	STP.P210A3_LimePumpS1_LocalRemoteStat AT %IX259.1 : BOOL;	(*  ~ {LinkedWith:TIID^C6920 (EtherCAT)^ScadaRoom_KouplerUTP (EK1100)^ScadaRoom_KouplerFiber (EK1521)^ChemicalAndTertiary (EK1501)^Term 90 (EL1809) A9^Channel 3^Input} *)
	STP.P203A_LimeCirculationPump1_LocalRemoteStat AT %IX111.1 : BOOL;	(*  ~ {LinkedWith:TIID^C6920 (EtherCAT)^ScadaRoom_KouplerUTP (EK1100)^ScadaRoom_KouplerFiber (EK1521)^ChemicalAndTertiary (EK1501)^Term 90 (EL1809) A9^Channel 6^Input} *)
	STP.P203B_LimeCirculationPump2_LocalRemoteStat AT %IX259.2 : BOOL;	(*  ~ {LinkedWith:TIID^C6920 (EtherCAT)^ScadaRoom_KouplerUTP (EK1100)^ScadaRoom_KouplerFiber (EK1521)^ChemicalAndTertiary (EK1501)^Term 90 (EL1809) A9^Channel 7^Input} *)
	STP.P211A1_AlumPumpSBRS1_LocalRemoteStat AT %IX96.1 : BOOL;	(*  ~ {LinkedWith:TIID^C6920 (EtherCAT)^ScadaRoom_KouplerUTP (EK1100)^ScadaRoom_KouplerFiber (EK1521)^ChemicalAndTertiary (EK1501)^Term 90 (EL1809) A9^Channel 8^Input} *)
	STP.P211A2_AlumPumpSBRS1_LocalRemoteStat AT %IX96.2 : BOOL;	(*  ~ {LinkedWith:TIID^C6920 (EtherCAT)^ScadaRoom_KouplerUTP (EK1100)^ScadaRoom_KouplerFiber (EK1521)^ChemicalAndTertiary (EK1501)^Term 90 (EL1809) A9^Channel 9^Input} *)
	STP.P211B1_AlumPumpSBRS2_LocalRemoteStat AT %IX96.3 : BOOL;	(*  ~ {LinkedWith:TIID^C6920 (EtherCAT)^ScadaRoom_KouplerUTP (EK1100)^ScadaRoom_KouplerFiber (EK1521)^ChemicalAndTertiary (EK1501)^Term 90 (EL1809) A9^Channel 10^Input} *)
	STP.P211B2_AlumPump2SBRS2_LocalRemoteStat AT %IX96.4 : BOOL;	(*  ~ {LinkedWith:TIID^C6920 (EtherCAT)^ScadaRoom_KouplerUTP (EK1100)^ScadaRoom_KouplerFiber (EK1521)^ChemicalAndTertiary (EK1501)^Term 90 (EL1809) A9^Channel 11^Input} *)
	STP.P352A_AlumPumpTertiaryDosing_LocalRemoteStat AT %IX111.2 : BOOL;	(*  ~ {LinkedWith:TIID^C6920 (EtherCAT)^ScadaRoom_KouplerUTP (EK1100)^ScadaRoom_KouplerFiber (EK1521)^ChemicalAndTertiary (EK1501)^Term 90 (EL1809) A9^Channel 12^Input} *)
	STP.P352B_AlumPumpTertiaryDosing_LocalRemoteStat AT %IX111.3 : BOOL;	(*  ~ {LinkedWith:TIID^C6920 (EtherCAT)^ScadaRoom_KouplerUTP (EK1100)^ScadaRoom_KouplerFiber (EK1521)^ChemicalAndTertiary (EK1501)^Term 90 (EL1809) A9^Channel 13^Input} *)
	STP.P354A_CausticSodaPump_LocalRemoteStat AT %IX111.4 : BOOL;	(*  ~ {LinkedWith:TIID^C6920 (EtherCAT)^ScadaRoom_KouplerUTP (EK1100)^ScadaRoom_KouplerFiber (EK1521)^ChemicalAndTertiary (EK1501)^Term 90 (EL1809) A9^Channel 14^Input} *)
	STP.P354B_CausticSodaPump_LocalRemoteStat AT %IX111.5 : BOOL;	(*  ~ {LinkedWith:TIID^C6920 (EtherCAT)^ScadaRoom_KouplerUTP (EK1100)^ScadaRoom_KouplerFiber (EK1521)^ChemicalAndTertiary (EK1501)^Term 90 (EL1809) A9^Channel 15^Input} *)
	STP.P356A_SodiumHypochloritePump_LocalRemoteStat AT %IX112.0 : BOOL;	(*  ~ {LinkedWith:TIID^C6920 (EtherCAT)^ScadaRoom_KouplerUTP (EK1100)^ScadaRoom_KouplerFiber (EK1521)^ChemicalAndTertiary (EK1501)^Term 91 (EL1809) A10^Channel 3^Input} *)
	STP.P356B_SodiumHypochloritePump_LocalRemoteStat AT %IX112.1 : BOOL;	(*  ~ {LinkedWith:TIID^C6920 (EtherCAT)^ScadaRoom_KouplerUTP (EK1100)^ScadaRoom_KouplerFiber (EK1521)^ChemicalAndTertiary (EK1501)^Term 91 (EL1809) A10^Channel 4^Input} *)
	STP.P301A_EffluentTransferPump_LocalRemoteStat AT %IX112.2 : BOOL;	(*  ~ {LinkedWith:TIID^C6920 (EtherCAT)^ScadaRoom_KouplerUTP (EK1100)^ScadaRoom_KouplerFiber (EK1521)^ChemicalAndTertiary (EK1501)^Term 91 (EL1809) A10^Channel 5^Input} *)
	STP.P301B_EffluentTransferPump_LocalRemoteStat AT %IX112.3 : BOOL;	(*  ~ {LinkedWith:TIID^C6920 (EtherCAT)^ScadaRoom_KouplerUTP (EK1100)^ScadaRoom_KouplerFiber (EK1521)^ChemicalAndTertiary (EK1501)^Term 91 (EL1809) A10^Channel 6^Input} *)
	STP.P302A_CollectionPump_LocalRemoteStat AT %IX112.4 : BOOL;	(*  ~ {LinkedWith:TIID^C6920 (EtherCAT)^ScadaRoom_KouplerUTP (EK1100)^ScadaRoom_KouplerFiber (EK1521)^ChemicalAndTertiary (EK1501)^Term 91 (EL1809) A10^Channel 7^Input} *)
	STP.P302B_CollectionPump_LocalRemoteStat AT %IX112.5 : BOOL;	(*  ~ {LinkedWith:TIID^C6920 (EtherCAT)^ScadaRoom_KouplerUTP (EK1100)^ScadaRoom_KouplerFiber (EK1521)^ChemicalAndTertiary (EK1501)^Term 91 (EL1809) A10^Channel 8^Input} *)
	STP.K301A_AirCompressor_LocalRemoteStat AT %IX112.6 : BOOL;	(*  ~ {LinkedWith:TIID^C6920 (EtherCAT)^ScadaRoom_KouplerUTP (EK1100)^ScadaRoom_KouplerFiber (EK1521)^ChemicalAndTertiary (EK1501)^Term 91 (EL1809) A10^Channel 9^Input} *)
	STP.K301B_AirCompressor_LocalRemoteStat AT %IX112.7 : BOOL;	(*  ~ {LinkedWith:TIID^C6920 (EtherCAT)^ScadaRoom_KouplerUTP (EK1100)^ScadaRoom_KouplerFiber (EK1521)^ChemicalAndTertiary (EK1501)^Term 91 (EL1809) A10^Channel 10^Input} *)
	STP.M210A_LimeStirrer_LocalRemoteStat AT %IX288.0 : BOOL;	(*  ~ {LinkedWith:TIID^C6920 (EtherCAT)^ScadaRoom_KouplerUTP (EK1100)^ScadaRoom_KouplerFiber (EK1521)^ChemicalAndTertiary (EK1501)^Term 91 (EL1809) A10^Channel 11^Input} *)
	STP.M210B_LimeStirrer_LocalRemoteStat AT %IX288.1 : BOOL;	(*  ~ {LinkedWith:TIID^C6920 (EtherCAT)^ScadaRoom_KouplerUTP (EK1100)^ScadaRoom_KouplerFiber (EK1521)^ChemicalAndTertiary (EK1501)^Term 91 (EL1809) A10^Channel 12^Input} *)
	STP.M210C_LimeStirrer_LocalRemoteStat AT %IX288.2 : BOOL;	(*  ~ {LinkedWith:TIID^C6920 (EtherCAT)^ScadaRoom_KouplerUTP (EK1100)^ScadaRoom_KouplerFiber (EK1521)^ChemicalAndTertiary (EK1501)^Term 91 (EL1809) A10^Channel 13^Input} *)
	STP.P210A1_LimePumpS1_TripStat AT %IX113.0 : BOOL;	(*  ~ {LinkedWith:TIID^C6920 (EtherCAT)^ScadaRoom_KouplerUTP (EK1100)^ScadaRoom_KouplerFiber (EK1521)^ChemicalAndTertiary (EK1501)^Term 92 (EL1809) A11^Channel 1^Input} *)
	STP.P210A2_LimePumpS1_TripStat AT %IX113.1 : BOOL;	(*  ~ {LinkedWith:TIID^C6920 (EtherCAT)^ScadaRoom_KouplerUTP (EK1100)^ScadaRoom_KouplerFiber (EK1521)^ChemicalAndTertiary (EK1501)^Term 92 (EL1809) A11^Channel 2^Input} *)
	STP.P210A3_LimePumpS1_TripStat AT %IX113.2 : BOOL;	(*  ~ {LinkedWith:TIID^C6920 (EtherCAT)^ScadaRoom_KouplerUTP (EK1100)^ScadaRoom_KouplerFiber (EK1521)^ChemicalAndTertiary (EK1501)^Term 92 (EL1809) A11^Channel 3^Input} *)
	STP.P203A_LimeCirculationPump_TripStat AT %IX113.3 : BOOL;	(*  ~ {LinkedWith:TIID^C6920 (EtherCAT)^ScadaRoom_KouplerUTP (EK1100)^ScadaRoom_KouplerFiber (EK1521)^ChemicalAndTertiary (EK1501)^Term 92 (EL1809) A11^Channel 6^Input} *)
	STP.P203B_LimeCirculationPump_TripStat AT %IX113.4 : BOOL;	(*  ~ {LinkedWith:TIID^C6920 (EtherCAT)^ScadaRoom_KouplerUTP (EK1100)^ScadaRoom_KouplerFiber (EK1521)^ChemicalAndTertiary (EK1501)^Term 92 (EL1809) A11^Channel 7^Input} *)
	STP.P211A1_AlumPumpSBRS1_TripStat AT %IX113.5 : BOOL;	(*  ~ {LinkedWith:TIID^C6920 (EtherCAT)^ScadaRoom_KouplerUTP (EK1100)^ScadaRoom_KouplerFiber (EK1521)^ChemicalAndTertiary (EK1501)^Term 92 (EL1809) A11^Channel 8^Input} *)
	STP.P211A2_AlumPumpSBRS1_TripStat AT %IX113.6 : BOOL;	(*  ~ {LinkedWith:TIID^C6920 (EtherCAT)^ScadaRoom_KouplerUTP (EK1100)^ScadaRoom_KouplerFiber (EK1521)^ChemicalAndTertiary (EK1501)^Term 92 (EL1809) A11^Channel 9^Input} *)
	STP.P211B1_AlumPumpSBRS1_TripStat AT %IX113.7 : BOOL;	(*  ~ {LinkedWith:TIID^C6920 (EtherCAT)^ScadaRoom_KouplerUTP (EK1100)^ScadaRoom_KouplerFiber (EK1521)^ChemicalAndTertiary (EK1501)^Term 92 (EL1809) A11^Channel 10^Input} *)
	STP.P211B2_AlumPumpSBRS2_TripStat AT %IX114.0 : BOOL;	(*  ~ {LinkedWith:TIID^C6920 (EtherCAT)^ScadaRoom_KouplerUTP (EK1100)^ScadaRoom_KouplerFiber (EK1521)^ChemicalAndTertiary (EK1501)^Term 92 (EL1809) A11^Channel 11^Input} *)
	STP.P352A_AlumPumpTertiaryDosing_TripStat AT %IX114.1 : BOOL;	(*  ~ {LinkedWith:TIID^C6920 (EtherCAT)^ScadaRoom_KouplerUTP (EK1100)^ScadaRoom_KouplerFiber (EK1521)^ChemicalAndTertiary (EK1501)^Term 92 (EL1809) A11^Channel 12^Input} *)
	STP.P352B_AlumPumpTertiaryDosing_TripStat AT %IX114.2 : BOOL;	(*  ~ {LinkedWith:TIID^C6920 (EtherCAT)^ScadaRoom_KouplerUTP (EK1100)^ScadaRoom_KouplerFiber (EK1521)^ChemicalAndTertiary (EK1501)^Term 92 (EL1809) A11^Channel 13^Input} *)
	STP.P354A_CausticSodaPump_TripStat AT %IX114.3 : BOOL;	(*  ~ {LinkedWith:TIID^C6920 (EtherCAT)^ScadaRoom_KouplerUTP (EK1100)^ScadaRoom_KouplerFiber (EK1521)^ChemicalAndTertiary (EK1501)^Term 92 (EL1809) A11^Channel 14^Input} *)
	STP.P354B_CausticSodaPump_TripStat AT %IX114.4 : BOOL;	(*  ~ {LinkedWith:TIID^C6920 (EtherCAT)^ScadaRoom_KouplerUTP (EK1100)^ScadaRoom_KouplerFiber (EK1521)^ChemicalAndTertiary (EK1501)^Term 92 (EL1809) A11^Channel 15^Input} *)
	STP.P356A_SodiumHypochloritePump_TripStat AT %IX114.7 : BOOL;	(*  ~ {LinkedWith:TIID^C6920 (EtherCAT)^ScadaRoom_KouplerUTP (EK1100)^ScadaRoom_KouplerFiber (EK1521)^ChemicalAndTertiary (EK1501)^Term 93 (EL1809) A12^Channel 3^Input} *)
	STP.P356B_SodiumHypochloritePump_TripStat AT %IX115.0 : BOOL;	(*  ~ {LinkedWith:TIID^C6920 (EtherCAT)^ScadaRoom_KouplerUTP (EK1100)^ScadaRoom_KouplerFiber (EK1521)^ChemicalAndTertiary (EK1501)^Term 93 (EL1809) A12^Channel 4^Input} *)
	STP.P301A_EffluentTransferPump_TripStat AT %IX115.1 : BOOL;	(*  ~ {LinkedWith:TIID^C6920 (EtherCAT)^ScadaRoom_KouplerUTP (EK1100)^ScadaRoom_KouplerFiber (EK1521)^ChemicalAndTertiary (EK1501)^Term 93 (EL1809) A12^Channel 5^Input} *)
	STP.P301B_EffluentTransferPump_TripStat AT %IX115.2 : BOOL;	(*  ~ {LinkedWith:TIID^C6920 (EtherCAT)^ScadaRoom_KouplerUTP (EK1100)^ScadaRoom_KouplerFiber (EK1521)^ChemicalAndTertiary (EK1501)^Term 93 (EL1809) A12^Channel 6^Input} *)
	STP.P302A_CollectionPump_TripStat AT %IX115.3 : BOOL;	(*  ~ {LinkedWith:TIID^C6920 (EtherCAT)^ScadaRoom_KouplerUTP (EK1100)^ScadaRoom_KouplerFiber (EK1521)^ChemicalAndTertiary (EK1501)^Term 93 (EL1809) A12^Channel 7^Input} *)
	STP.P302B_CollectionPump_TripStat AT %IX115.4 : BOOL;	(*  ~ {LinkedWith:TIID^C6920 (EtherCAT)^ScadaRoom_KouplerUTP (EK1100)^ScadaRoom_KouplerFiber (EK1521)^ChemicalAndTertiary (EK1501)^Term 93 (EL1809) A12^Channel 8^Input} *)
	STP.K301A_AirCompressor_TripStat AT %IX115.5 : BOOL;	(*  ~ {LinkedWith:TIID^C6920 (EtherCAT)^ScadaRoom_KouplerUTP (EK1100)^ScadaRoom_KouplerFiber (EK1521)^ChemicalAndTertiary (EK1501)^Term 93 (EL1809) A12^Channel 9^Input} *)
	STP.K301B_AirCompressor_TripStat AT %IX115.6 : BOOL;	(*  ~ {LinkedWith:TIID^C6920 (EtherCAT)^ScadaRoom_KouplerUTP (EK1100)^ScadaRoom_KouplerFiber (EK1521)^ChemicalAndTertiary (EK1501)^Term 93 (EL1809) A12^Channel 10^Input} *)
	STP.M303A_Floculator_TripStat AT %IX259.3 : BOOL;	(*  ~ {LinkedWith:TIID^C6920 (EtherCAT)^ScadaRoom_KouplerUTP (EK1100)^ScadaRoom_KouplerFiber (EK1521)^ChemicalAndTertiary (EK1501)^Term 93 (EL1809) A12^Channel 11^Input} *)
	STP.M303B_Floculator_TripStat AT %IX259.4 : BOOL;	(*  ~ {LinkedWith:TIID^C6920 (EtherCAT)^ScadaRoom_KouplerUTP (EK1100)^ScadaRoom_KouplerFiber (EK1521)^ChemicalAndTertiary (EK1501)^Term 93 (EL1809) A12^Channel 12^Input} *)
	STP.M303C_Floculator_TripStat AT %IX259.5 : BOOL;	(*  ~ {LinkedWith:TIID^C6920 (EtherCAT)^ScadaRoom_KouplerUTP (EK1100)^ScadaRoom_KouplerFiber (EK1521)^ChemicalAndTertiary (EK1501)^Term 93 (EL1809) A12^Channel 13^Input} *)
	STP.M303D_Floculator_TripStat AT %IX259.6 : BOOL;	(*  ~ {LinkedWith:TIID^C6920 (EtherCAT)^ScadaRoom_KouplerUTP (EK1100)^ScadaRoom_KouplerFiber (EK1521)^ChemicalAndTertiary (EK1501)^Term 93 (EL1809) A12^Channel 14^Input} *)
	STP.P210A1_LimePumpS1_EStopStat AT %IX259.7 : BOOL;	(*  ~ {LinkedWith:TIID^C6920 (EtherCAT)^ScadaRoom_KouplerUTP (EK1100)^ScadaRoom_KouplerFiber (EK1521)^ChemicalAndTertiary (EK1501)^Term 94 (EL1809) A13^Channel 1^Input} *)
	STP.P210A2_LimePumpS1_EStopStat AT %IX260.0 : BOOL;	(*  ~ {LinkedWith:TIID^C6920 (EtherCAT)^ScadaRoom_KouplerUTP (EK1100)^ScadaRoom_KouplerFiber (EK1521)^ChemicalAndTertiary (EK1501)^Term 94 (EL1809) A13^Channel 2^Input} *)
	STP.P210A3_LimePumpS1_EStopStat AT %IX260.1 : BOOL;	(*  ~ {LinkedWith:TIID^C6920 (EtherCAT)^ScadaRoom_KouplerUTP (EK1100)^ScadaRoom_KouplerFiber (EK1521)^ChemicalAndTertiary (EK1501)^Term 94 (EL1809) A13^Channel 3^Input} *)
	STP.P203A_LimeCirculationPump_EStopStat AT %IX260.2 : BOOL;	(*  ~ {LinkedWith:TIID^C6920 (EtherCAT)^ScadaRoom_KouplerUTP (EK1100)^ScadaRoom_KouplerFiber (EK1521)^ChemicalAndTertiary (EK1501)^Term 94 (EL1809) A13^Channel 6^Input} *)
	STP.P203B_LimeCirculationPump_EStopStat AT %IX260.3 : BOOL;	(*  ~ {LinkedWith:TIID^C6920 (EtherCAT)^ScadaRoom_KouplerUTP (EK1100)^ScadaRoom_KouplerFiber (EK1521)^ChemicalAndTertiary (EK1501)^Term 94 (EL1809) A13^Channel 7^Input} *)
	STP.P211A1_AlumPumpSBRS1_EStopStat AT %IX260.4 : BOOL;	(*  ~ {LinkedWith:TIID^C6920 (EtherCAT)^ScadaRoom_KouplerUTP (EK1100)^ScadaRoom_KouplerFiber (EK1521)^ChemicalAndTertiary (EK1501)^Term 94 (EL1809) A13^Channel 8^Input} *)
	STP.P211A2_AlumPumpSBRS1_EStopStat AT %IX260.5 : BOOL;	(*  ~ {LinkedWith:TIID^C6920 (EtherCAT)^ScadaRoom_KouplerUTP (EK1100)^ScadaRoom_KouplerFiber (EK1521)^ChemicalAndTertiary (EK1501)^Term 94 (EL1809) A13^Channel 9^Input} *)
	STP.P211B1_AlumPumpSBRS2_EStopStat AT %IX260.6 : BOOL;	(*  ~ {LinkedWith:TIID^C6920 (EtherCAT)^ScadaRoom_KouplerUTP (EK1100)^ScadaRoom_KouplerFiber (EK1521)^ChemicalAndTertiary (EK1501)^Term 94 (EL1809) A13^Channel 10^Input} *)
	STP.P211B2_AlumPumpSBRS2_EStopStat AT %IX260.7 : BOOL;	(*  ~ {LinkedWith:TIID^C6920 (EtherCAT)^ScadaRoom_KouplerUTP (EK1100)^ScadaRoom_KouplerFiber (EK1521)^ChemicalAndTertiary (EK1501)^Term 94 (EL1809) A13^Channel 11^Input} *)
	STP.P352A_AlumPumpTertiaryDosing_EStopStat AT %IX261.0 : BOOL;	(*  ~ {LinkedWith:TIID^C6920 (EtherCAT)^ScadaRoom_KouplerUTP (EK1100)^ScadaRoom_KouplerFiber (EK1521)^ChemicalAndTertiary (EK1501)^Term 94 (EL1809) A13^Channel 12^Input} *)
	STP.P352B_AlumPumpTertiaryDosing_EStopStat AT %IX261.1 : BOOL;	(*  ~ {LinkedWith:TIID^C6920 (EtherCAT)^ScadaRoom_KouplerUTP (EK1100)^ScadaRoom_KouplerFiber (EK1521)^ChemicalAndTertiary (EK1501)^Term 94 (EL1809) A13^Channel 13^Input} *)
	STP.P354A_CausticSodaPump_EStopStat AT %IX261.2 : BOOL;	(*  ~ {LinkedWith:TIID^C6920 (EtherCAT)^ScadaRoom_KouplerUTP (EK1100)^ScadaRoom_KouplerFiber (EK1521)^ChemicalAndTertiary (EK1501)^Term 94 (EL1809) A13^Channel 14^Input} *)
	STP.P354B_CausticSodaPump_EStopStat AT %IX261.3 : BOOL;	(*  ~ {LinkedWith:TIID^C6920 (EtherCAT)^ScadaRoom_KouplerUTP (EK1100)^ScadaRoom_KouplerFiber (EK1521)^ChemicalAndTertiary (EK1501)^Term 94 (EL1809) A13^Channel 15^Input} *)
	STP.P356A_SodiumHypochloritePump_EStopStat AT %IX261.4 : BOOL;	(*  ~ {LinkedWith:TIID^C6920 (EtherCAT)^ScadaRoom_KouplerUTP (EK1100)^ScadaRoom_KouplerFiber (EK1521)^ChemicalAndTertiary (EK1501)^Term 95 (EL1809) A14^Channel 3^Input} *)
	STP.P356B_SodiumHypochloritePump_EStopStat AT %IX261.5 : BOOL;	(*  ~ {LinkedWith:TIID^C6920 (EtherCAT)^ScadaRoom_KouplerUTP (EK1100)^ScadaRoom_KouplerFiber (EK1521)^ChemicalAndTertiary (EK1501)^Term 95 (EL1809) A14^Channel 4^Input} *)
	STP.P301A_EffluentTransferPump_EStopStat AT %IX261.6 : BOOL;	(*  ~ {LinkedWith:TIID^C6920 (EtherCAT)^ScadaRoom_KouplerUTP (EK1100)^ScadaRoom_KouplerFiber (EK1521)^ChemicalAndTertiary (EK1501)^Term 95 (EL1809) A14^Channel 5^Input} *)
	STP.P301B_EffluentTransferPump_EStopStat AT %IX261.7 : BOOL;	(*  ~ {LinkedWith:TIID^C6920 (EtherCAT)^ScadaRoom_KouplerUTP (EK1100)^ScadaRoom_KouplerFiber (EK1521)^ChemicalAndTertiary (EK1501)^Term 95 (EL1809) A14^Channel 6^Input} *)
	STP.P302A_CollectionPump_EStopStat AT %IX262.0 : BOOL;	(*  ~ {LinkedWith:TIID^C6920 (EtherCAT)^ScadaRoom_KouplerUTP (EK1100)^ScadaRoom_KouplerFiber (EK1521)^ChemicalAndTertiary (EK1501)^Term 95 (EL1809) A14^Channel 7^Input} *)
	STP.P302B_CollectionPump_EStopStat AT %IX262.1 : BOOL;	(*  ~ {LinkedWith:TIID^C6920 (EtherCAT)^ScadaRoom_KouplerUTP (EK1100)^ScadaRoom_KouplerFiber (EK1521)^ChemicalAndTertiary (EK1501)^Term 95 (EL1809) A14^Channel 8^Input} *)
	STP.K301A_AirCompressor_EStopStat AT %IX262.2 : BOOL;	(*  ~ {LinkedWith:TIID^C6920 (EtherCAT)^ScadaRoom_KouplerUTP (EK1100)^ScadaRoom_KouplerFiber (EK1521)^ChemicalAndTertiary (EK1501)^Term 95 (EL1809) A14^Channel 9^Input} *)
	STP.K301B_AirCompressor_EStopStat AT %IX262.3 : BOOL;	(*  ~ {LinkedWith:TIID^C6920 (EtherCAT)^ScadaRoom_KouplerUTP (EK1100)^ScadaRoom_KouplerFiber (EK1521)^ChemicalAndTertiary (EK1501)^Term 95 (EL1809) A14^Channel 10^Input} *)
	STP.M210A_LimeStirrer_EStopStat AT %IX288.3 : BOOL;	(*  ~ {LinkedWith:TIID^C6920 (EtherCAT)^ScadaRoom_KouplerUTP (EK1100)^ScadaRoom_KouplerFiber (EK1521)^ChemicalAndTertiary (EK1501)^Term 95 (EL1809) A14^Channel 11^Input} *)
	STP.M210B_LimeStirrer_EStopStat AT %IX288.4 : BOOL;	(*  ~ {LinkedWith:TIID^C6920 (EtherCAT)^ScadaRoom_KouplerUTP (EK1100)^ScadaRoom_KouplerFiber (EK1521)^ChemicalAndTertiary (EK1501)^Term 95 (EL1809) A14^Channel 12^Input} *)
	STP.M210C_LimeStirrer_EStopStat AT %IX288.5 : BOOL;	(*  ~ {LinkedWith:TIID^C6920 (EtherCAT)^ScadaRoom_KouplerUTP (EK1100)^ScadaRoom_KouplerFiber (EK1521)^ChemicalAndTertiary (EK1501)^Term 95 (EL1809) A14^Channel 13^Input} *)
	STP.XV250A_LimeWaterIntakeTank_OpenCmd AT %QX40.0 : BOOL;	(*  ~ {LinkedWith:TIID^C6920 (EtherCAT)^ScadaRoom_KouplerUTP (EK1100)^ScadaRoom_KouplerFiber (EK1521)^ChemicalAndTertiary (EK1501)^Term 96 (EK1122)^Term 97 (EK1100)^Term 98 (EL2809) A18^Channel 1^Output} *)
	STP.XV250B_LimeWaterIntakeTank_OpenCmd AT %QX59.3 : BOOL;	(*  ~ {LinkedWith:TIID^C6920 (EtherCAT)^ScadaRoom_KouplerUTP (EK1100)^ScadaRoom_KouplerFiber (EK1521)^ChemicalAndTertiary (EK1501)^Term 96 (EK1122)^Term 97 (EK1100)^Term 98 (EL2809) A18^Channel 2^Output} *)
	STP.XV250C_LimeWaterIntakeTank_OpenCmd AT %QX40.2 : BOOL;	(*  ~ {LinkedWith:TIID^C6920 (EtherCAT)^ScadaRoom_KouplerUTP (EK1100)^ScadaRoom_KouplerFiber (EK1521)^ChemicalAndTertiary (EK1501)^Term 96 (EK1122)^Term 97 (EK1100)^Term 98 (EL2809) A18^Channel 3^Output} *)
	STP.XV251A_LimeSelectorTank_OpenCmd AT %QX40.3 : BOOL;	(*  ~ {LinkedWith:TIID^C6920 (EtherCAT)^ScadaRoom_KouplerUTP (EK1100)^ScadaRoom_KouplerFiber (EK1521)^ChemicalAndTertiary (EK1501)^Term 96 (EK1122)^Term 97 (EK1100)^Term 98 (EL2809) A18^Channel 4^Output} *)
	STP.XV251B_LimeSelectorTank_OpenCmd AT %QX40.4 : BOOL;	(*  ~ {LinkedWith:TIID^C6920 (EtherCAT)^ScadaRoom_KouplerUTP (EK1100)^ScadaRoom_KouplerFiber (EK1521)^ChemicalAndTertiary (EK1501)^Term 96 (EK1122)^Term 97 (EK1100)^Term 98 (EL2809) A18^Channel 5^Output} *)
	STP.XV251C_LimeSelectorTank_OpenCmd AT %QX40.5 : BOOL;	(*  ~ {LinkedWith:TIID^C6920 (EtherCAT)^ScadaRoom_KouplerUTP (EK1100)^ScadaRoom_KouplerFiber (EK1521)^ChemicalAndTertiary (EK1501)^Term 96 (EK1122)^Term 97 (EK1100)^Term 98 (EL2809) A18^Channel 6^Output} *)
	STP.M210A_LimeStirrer_RunCmd AT %QX76.0 : BOOL;	(*  ~ {LinkedWith:TIID^C6920 (EtherCAT)^ScadaRoom_KouplerUTP (EK1100)^ScadaRoom_KouplerFiber (EK1521)^ChemicalAndTertiary (EK1501)^Term 96 (EK1122)^Term 97 (EK1100)^Term 98 (EL2809) A18^Channel 7^Output} *)
	STP.M210B_LimeStirrer_RunCmd AT %QX76.1 : BOOL;	(*  ~ {LinkedWith:TIID^C6920 (EtherCAT)^ScadaRoom_KouplerUTP (EK1100)^ScadaRoom_KouplerFiber (EK1521)^ChemicalAndTertiary (EK1501)^Term 96 (EK1122)^Term 97 (EK1100)^Term 98 (EL2809) A18^Channel 8^Output} *)
	STP.M210C_LimeStirrer_RunCmd AT %QX76.2 : BOOL;	(*  ~ {LinkedWith:TIID^C6920 (EtherCAT)^ScadaRoom_KouplerUTP (EK1100)^ScadaRoom_KouplerFiber (EK1521)^ChemicalAndTertiary (EK1501)^Term 96 (EK1122)^Term 97 (EK1100)^Term 98 (EL2809) A18^Channel 9^Output} *)
	STP.P210A1_LimePumpS1_RunCmd AT %QX59.4 : BOOL;	(*  ~ {LinkedWith:TIID^C6920 (EtherCAT)^ScadaRoom_KouplerUTP (EK1100)^ScadaRoom_KouplerFiber (EK1521)^ChemicalAndTertiary (EK1501)^Term 96 (EK1122)^Term 97 (EK1100)^Term 98 (EL2809) A18^Channel 10^Output} *)
	STP.P210A2_LimePumpS1_RunCmd AT %QX59.5 : BOOL;	(*  ~ {LinkedWith:TIID^C6920 (EtherCAT)^ScadaRoom_KouplerUTP (EK1100)^ScadaRoom_KouplerFiber (EK1521)^ChemicalAndTertiary (EK1501)^Term 96 (EK1122)^Term 97 (EK1100)^Term 98 (EL2809) A18^Channel 11^Output} *)
	STP.P210A3_LimePumpS1_RunCmd AT %QX59.6 : BOOL;	(*  ~ {LinkedWith:TIID^C6920 (EtherCAT)^ScadaRoom_KouplerUTP (EK1100)^ScadaRoom_KouplerFiber (EK1521)^ChemicalAndTertiary (EK1501)^Term 96 (EK1122)^Term 97 (EK1100)^Term 98 (EL2809) A18^Channel 12^Output} *)
	STP.P210A1_LimeValveS2_OpenCmd AT %QX41.4 : BOOL;	(*  ~ {LinkedWith:TIID^C6920 (EtherCAT)^ScadaRoom_KouplerUTP (EK1100)^ScadaRoom_KouplerFiber (EK1521)^ChemicalAndTertiary (EK1501)^Term 96 (EK1122)^Term 97 (EK1100)^Term 98 (EL2809) A18^Channel 13^Output} *)
	STP.P210A2_LimeValveS2_OpenCmd AT %QX41.5 : BOOL;	(*  ~ {LinkedWith:TIID^C6920 (EtherCAT)^ScadaRoom_KouplerUTP (EK1100)^ScadaRoom_KouplerFiber (EK1521)^ChemicalAndTertiary (EK1501)^Term 96 (EK1122)^Term 97 (EK1100)^Term 98 (EL2809) A18^Channel 14^Output} *)
	STP.P354A_CausticSodaPump_RunCmd AT %QX42.0 : BOOL;	(*  ~ {LinkedWith:TIID^C6920 (EtherCAT)^ScadaRoom_KouplerUTP (EK1100)^ScadaRoom_KouplerFiber (EK1521)^ChemicalAndTertiary (EK1501)^Term 96 (EK1122)^Term 97 (EK1100)^Term 99 (EL2809) A19^Channel 1^Output} *)
	STP.P354B_CausticSodaPump_RunCmd AT %QX42.1 : BOOL;	(*  ~ {LinkedWith:TIID^C6920 (EtherCAT)^ScadaRoom_KouplerUTP (EK1100)^ScadaRoom_KouplerFiber (EK1521)^ChemicalAndTertiary (EK1501)^Term 96 (EK1122)^Term 97 (EK1100)^Term 99 (EL2809) A19^Channel 2^Output} *)
	STP.P356A_SodiumHypochloritePump_RunCmd AT %QX42.2 : BOOL;	(*  ~ {LinkedWith:TIID^C6920 (EtherCAT)^ScadaRoom_KouplerUTP (EK1100)^ScadaRoom_KouplerFiber (EK1521)^ChemicalAndTertiary (EK1501)^Term 96 (EK1122)^Term 97 (EK1100)^Term 99 (EL2809) A19^Channel 3^Output} *)
	STP.P356B_SodiumHypochloritePump_RunCmd AT %QX42.3 : BOOL;	(*  ~ {LinkedWith:TIID^C6920 (EtherCAT)^ScadaRoom_KouplerUTP (EK1100)^ScadaRoom_KouplerFiber (EK1521)^ChemicalAndTertiary (EK1501)^Term 96 (EK1122)^Term 97 (EK1100)^Term 99 (EL2809) A19^Channel 4^Output} *)
	STP.P204A_SodiumHypochloritePump_RunCmd AT %QX42.4 : BOOL;	(*  ~ {LinkedWith:TIID^C6920 (EtherCAT)^ScadaRoom_KouplerUTP (EK1100)^ScadaRoom_KouplerFiber (EK1521)^ChemicalAndTertiary (EK1501)^Term 96 (EK1122)^Term 97 (EK1100)^Term 99 (EL2809) A19^Channel 5^Output} *)
	STP.P211A1_AlumPumpSBRS1_RunCmd AT %QX42.6 : BOOL;	(*  ~ {LinkedWith:TIID^C6920 (EtherCAT)^ScadaRoom_KouplerUTP (EK1100)^ScadaRoom_KouplerFiber (EK1521)^ChemicalAndTertiary (EK1501)^Term 96 (EK1122)^Term 97 (EK1100)^Term 99 (EL2809) A19^Channel 7^Output} *)
	STP.P211A2_AlumPumpSBRS1_RunCmd AT %QX42.7 : BOOL;	(*  ~ {LinkedWith:TIID^C6920 (EtherCAT)^ScadaRoom_KouplerUTP (EK1100)^ScadaRoom_KouplerFiber (EK1521)^ChemicalAndTertiary (EK1501)^Term 96 (EK1122)^Term 97 (EK1100)^Term 99 (EL2809) A19^Channel 8^Output} *)
	STP.P211B1_AlumPumpSBRS2_RunCmd AT %QX43.0 : BOOL;	(*  ~ {LinkedWith:TIID^C6920 (EtherCAT)^ScadaRoom_KouplerUTP (EK1100)^ScadaRoom_KouplerFiber (EK1521)^ChemicalAndTertiary (EK1501)^Term 96 (EK1122)^Term 97 (EK1100)^Term 99 (EL2809) A19^Channel 9^Output} *)
	STP.P211B2_AlumPumpSBRS2_RunCmd AT %QX43.1 : BOOL;	(*  ~ {LinkedWith:TIID^C6920 (EtherCAT)^ScadaRoom_KouplerUTP (EK1100)^ScadaRoom_KouplerFiber (EK1521)^ChemicalAndTertiary (EK1501)^Term 96 (EK1122)^Term 97 (EK1100)^Term 99 (EL2809) A19^Channel 10^Output} *)
	STP.P352A_AlumPumpTertiaryDosing_RunCmd AT %QX59.7 : BOOL;	(*  ~ {LinkedWith:TIID^C6920 (EtherCAT)^ScadaRoom_KouplerUTP (EK1100)^ScadaRoom_KouplerFiber (EK1521)^ChemicalAndTertiary (EK1501)^Term 96 (EK1122)^Term 97 (EK1100)^Term 99 (EL2809) A19^Channel 11^Output} *)
	STP.P352B_AlumPumpTertiaryDosing_RunCmd AT %QX60.0 : BOOL;	(*  ~ {LinkedWith:TIID^C6920 (EtherCAT)^ScadaRoom_KouplerUTP (EK1100)^ScadaRoom_KouplerFiber (EK1521)^ChemicalAndTertiary (EK1501)^Term 96 (EK1122)^Term 97 (EK1100)^Term 99 (EL2809) A19^Channel 12^Output} *)
	STP.P203A_LimeCirculationPump_RunCmd AT %QX43.4 : BOOL;	(*  ~ {LinkedWith:TIID^C6920 (EtherCAT)^ScadaRoom_KouplerUTP (EK1100)^ScadaRoom_KouplerFiber (EK1521)^ChemicalAndTertiary (EK1501)^Term 96 (EK1122)^Term 97 (EK1100)^Term 99 (EL2809) A19^Channel 13^Output} *)
	STP.P203B_LimeCirculationPump_RunCmd AT %QX43.5 : BOOL;	(*  ~ {LinkedWith:TIID^C6920 (EtherCAT)^ScadaRoom_KouplerUTP (EK1100)^ScadaRoom_KouplerFiber (EK1521)^ChemicalAndTertiary (EK1501)^Term 96 (EK1122)^Term 97 (EK1100)^Term 99 (EL2809) A19^Channel 14^Output} *)
	STP.XV303A_LamellaSludgeDischarge_RunCmd AT %QX60.1 : BOOL;	(*  ~ {LinkedWith:TIID^C6920 (EtherCAT)^ScadaRoom_KouplerUTP (EK1100)^ScadaRoom_KouplerFiber (EK1521)^ChemicalAndTertiary (EK1501)^Term 96 (EK1122)^Term 97 (EK1100)^Term 100 (EL2809) A20^Channel 1^Output} *)
	STP.XV303B_LamellaSludgeDischarge_RunCmd AT %QX60.2 : BOOL;	(*  ~ {LinkedWith:TIID^C6920 (EtherCAT)^ScadaRoom_KouplerUTP (EK1100)^ScadaRoom_KouplerFiber (EK1521)^ChemicalAndTertiary (EK1501)^Term 96 (EK1122)^Term 97 (EK1100)^Term 100 (EL2809) A20^Channel 2^Output} *)
	STP.XV303C_LamellaSludgeDischarge_RunCmd AT %QX60.3 : BOOL;	(*  ~ {LinkedWith:TIID^C6920 (EtherCAT)^ScadaRoom_KouplerUTP (EK1100)^ScadaRoom_KouplerFiber (EK1521)^ChemicalAndTertiary (EK1501)^Term 96 (EK1122)^Term 97 (EK1100)^Term 100 (EL2809) A20^Channel 3^Output} *)
	STP.XV303D_LamellaSludgeDischarge_RunCmd AT %QX60.4 : BOOL;	(*  ~ {LinkedWith:TIID^C6920 (EtherCAT)^ScadaRoom_KouplerUTP (EK1100)^ScadaRoom_KouplerFiber (EK1521)^ChemicalAndTertiary (EK1501)^Term 96 (EK1122)^Term 97 (EK1100)^Term 100 (EL2809) A20^Channel 4^Output} *)
	STP.XV305_TertiaryTreatmentMainValve_OpenCmd AT %QX60.5 : BOOL;	(*  ~ {LinkedWith:TIID^C6920 (EtherCAT)^ScadaRoom_KouplerUTP (EK1100)^ScadaRoom_KouplerFiber (EK1521)^ChemicalAndTertiary (EK1501)^Term 96 (EK1122)^Term 97 (EK1100)^Term 100 (EL2809) A20^Channel 5^Output} *)
	STP.M303A_Floculator_RunCmd AT %QX44.3 : BOOL;	(*  ~ {LinkedWith:TIID^C6920 (EtherCAT)^ScadaRoom_KouplerUTP (EK1100)^ScadaRoom_KouplerFiber (EK1521)^ChemicalAndTertiary (EK1501)^Term 96 (EK1122)^Term 97 (EK1100)^Term 100 (EL2809) A20^Channel 6^Output} *)
	STP.M303B_Floculator_RunCmd AT %QX44.4 : BOOL;	(*  ~ {LinkedWith:TIID^C6920 (EtherCAT)^ScadaRoom_KouplerUTP (EK1100)^ScadaRoom_KouplerFiber (EK1521)^ChemicalAndTertiary (EK1501)^Term 96 (EK1122)^Term 97 (EK1100)^Term 100 (EL2809) A20^Channel 7^Output} *)
	STP.M303C_Floculator_RunCmd AT %QX44.5 : BOOL;	(*  ~ {LinkedWith:TIID^C6920 (EtherCAT)^ScadaRoom_KouplerUTP (EK1100)^ScadaRoom_KouplerFiber (EK1521)^ChemicalAndTertiary (EK1501)^Term 96 (EK1122)^Term 97 (EK1100)^Term 100 (EL2809) A20^Channel 8^Output} *)
	STP.M303D_Floculator_RunCmd AT %QX44.6 : BOOL;	(*  ~ {LinkedWith:TIID^C6920 (EtherCAT)^ScadaRoom_KouplerUTP (EK1100)^ScadaRoom_KouplerFiber (EK1521)^ChemicalAndTertiary (EK1501)^Term 96 (EK1122)^Term 97 (EK1100)^Term 100 (EL2809) A20^Channel 9^Output} *)
	STP.P301A_EffluentTransferPump_RunCmd AT %QX44.7 : BOOL;	(*  ~ {LinkedWith:TIID^C6920 (EtherCAT)^ScadaRoom_KouplerUTP (EK1100)^ScadaRoom_KouplerFiber (EK1521)^ChemicalAndTertiary (EK1501)^Term 96 (EK1122)^Term 97 (EK1100)^Term 100 (EL2809) A20^Channel 10^Output} *)
	STP.P301B_EffluentTransferPump_RunCmd AT %QX45.0 : BOOL;	(*  ~ {LinkedWith:TIID^C6920 (EtherCAT)^ScadaRoom_KouplerUTP (EK1100)^ScadaRoom_KouplerFiber (EK1521)^ChemicalAndTertiary (EK1501)^Term 96 (EK1122)^Term 97 (EK1100)^Term 100 (EL2809) A20^Channel 11^Output} *)
	STP.P302A_CollectionPump_RunCmd AT %QX45.1 : BOOL;	(*  ~ {LinkedWith:TIID^C6920 (EtherCAT)^ScadaRoom_KouplerUTP (EK1100)^ScadaRoom_KouplerFiber (EK1521)^ChemicalAndTertiary (EK1501)^Term 96 (EK1122)^Term 97 (EK1100)^Term 100 (EL2809) A20^Channel 12^Output} *)
	STP.P302B_CollectionPump_RunCmd AT %QX45.2 : BOOL;	(*  ~ {LinkedWith:TIID^C6920 (EtherCAT)^ScadaRoom_KouplerUTP (EK1100)^ScadaRoom_KouplerFiber (EK1521)^ChemicalAndTertiary (EK1501)^Term 96 (EK1122)^Term 97 (EK1100)^Term 100 (EL2809) A20^Channel 13^Output} *)
	STP.K301A_AirCompressor_RunCmd AT %QX45.3 : BOOL;	(*  ~ {LinkedWith:TIID^C6920 (EtherCAT)^ScadaRoom_KouplerUTP (EK1100)^ScadaRoom_KouplerFiber (EK1521)^ChemicalAndTertiary (EK1501)^Term 96 (EK1122)^Term 97 (EK1100)^Term 100 (EL2809) A20^Channel 14^Output} *)
	STP.K301B_AirCompressor_RunCmd AT %QX45.4 : BOOL;	(*  ~ {LinkedWith:TIID^C6920 (EtherCAT)^ScadaRoom_KouplerUTP (EK1100)^ScadaRoom_KouplerFiber (EK1521)^ChemicalAndTertiary (EK1501)^Term 96 (EK1122)^Term 97 (EK1100)^Term 100 (EL2809) A20^Channel 15^Output} *)
	STP.AUX1_CirculationOverflow AT %QX45.5 : BOOL;	(*  ~ {LinkedWith:TIID^C6920 (EtherCAT)^ScadaRoom_KouplerUTP (EK1100)^ScadaRoom_KouplerFiber (EK1521)^ChemicalAndTertiary (EK1501)^Term 96 (EK1122)^Term 97 (EK1100)^Term 101 (EL2809) A21^Channel 1^Output} *)
	STP.AUX2_SystemInletMonitoring AT %QX45.6 : BOOL;	(*  ~ {LinkedWith:TIID^C6920 (EtherCAT)^ScadaRoom_KouplerUTP (EK1100)^ScadaRoom_KouplerFiber (EK1521)^ChemicalAndTertiary (EK1501)^Term 96 (EK1122)^Term 97 (EK1100)^Term 101 (EL2809) A21^Channel 2^Output} *)
	STP.AUX3_SystemOutletMonitoring AT %QX45.7 : BOOL;	(*  ~ {LinkedWith:TIID^C6920 (EtherCAT)^ScadaRoom_KouplerUTP (EK1100)^ScadaRoom_KouplerFiber (EK1521)^ChemicalAndTertiary (EK1501)^Term 96 (EK1122)^Term 97 (EK1100)^Term 101 (EL2809) A21^Channel 3^Output} *)
	STP.AUX4_ChlorineHIGH AT %QX46.0 : BOOL;	(*  ~ {LinkedWith:TIID^C6920 (EtherCAT)^ScadaRoom_KouplerUTP (EK1100)^ScadaRoom_KouplerFiber (EK1521)^ChemicalAndTertiary (EK1501)^Term 96 (EK1122)^Term 97 (EK1100)^Term 101 (EL2809) A21^Channel 4^Output} *)
	STP.AUX5_SBRDosing AT %QX46.1 : BOOL;	(*  ~ {LinkedWith:TIID^C6920 (EtherCAT)^ScadaRoom_KouplerUTP (EK1100)^ScadaRoom_KouplerFiber (EK1521)^ChemicalAndTertiary (EK1501)^Term 96 (EK1122)^Term 97 (EK1100)^Term 101 (EL2809) A21^Channel 5^Output} *)
	STP.AUX6_ChlorineDosing AT %QX46.2 : BOOL;	(*  ~ {LinkedWith:TIID^C6920 (EtherCAT)^ScadaRoom_KouplerUTP (EK1100)^ScadaRoom_KouplerFiber (EK1521)^ChemicalAndTertiary (EK1501)^Term 96 (EK1122)^Term 97 (EK1100)^Term 101 (EL2809) A21^Channel 6^Output} *)
	STP.AUX7_DisinfectionDosing AT %QX46.3 : BOOL;	(*  ~ {LinkedWith:TIID^C6920 (EtherCAT)^ScadaRoom_KouplerUTP (EK1100)^ScadaRoom_KouplerFiber (EK1521)^ChemicalAndTertiary (EK1501)^Term 96 (EK1122)^Term 97 (EK1100)^Term 101 (EL2809) A21^Channel 7^Output} *)
	STP.AUX8_TertiaryDosing AT %QX46.4 : BOOL;	(*  ~ {LinkedWith:TIID^C6920 (EtherCAT)^ScadaRoom_KouplerUTP (EK1100)^ScadaRoom_KouplerFiber (EK1521)^ChemicalAndTertiary (EK1501)^Term 96 (EK1122)^Term 97 (EK1100)^Term 101 (EL2809) A21^Channel 8^Output} *)
	STP.AUX602_PLCRunStat AT %QX73.1 : BOOL;	(*  ~ {LinkedWith:TIID^C6920 (EtherCAT)^ScadaRoom_KouplerUTP (EK1100)^ScadaRoom_KouplerFiber (EK1521)^ChemicalAndTertiary (EK1501)^Term 96 (EK1122)^Term 97 (EK1100)^Term 101 (EL2809) A21^Channel 9^Output} *)
	STP.AUX601_CommonAlarm AT %QX73.2 : BOOL;	(*  ~ {LinkedWith:TIID^C6920 (EtherCAT)^ScadaRoom_KouplerUTP (EK1100)^ScadaRoom_KouplerFiber (EK1521)^ChemicalAndTertiary (EK1501)^Term 96 (EK1122)^Term 97 (EK1100)^Term 101 (EL2809) A21^Channel 10^Output} *)
	STP.AUX17_LimeInService AT %QX47.5 : BOOL;	(*  ~ {LinkedWith:TIID^C6920 (EtherCAT)^ScadaRoom_KouplerUTP (EK1100)^ScadaRoom_KouplerFiber (EK1521)^ChemicalAndTertiary (EK1501)^Term 96 (EK1122)^Term 97 (EK1100)^Term 102 (EL2809) A22^Channel 1^Output} *)
	STP.AUX18_LimeInService AT %QX47.6 : BOOL;	(*  ~ {LinkedWith:TIID^C6920 (EtherCAT)^ScadaRoom_KouplerUTP (EK1100)^ScadaRoom_KouplerFiber (EK1521)^ChemicalAndTertiary (EK1501)^Term 96 (EK1122)^Term 97 (EK1100)^Term 102 (EL2809) A22^Channel 2^Output} *)
	STP.AUX19_LimeInService AT %QX47.7 : BOOL;	(*  ~ {LinkedWith:TIID^C6920 (EtherCAT)^ScadaRoom_KouplerUTP (EK1100)^ScadaRoom_KouplerFiber (EK1521)^ChemicalAndTertiary (EK1501)^Term 96 (EK1122)^Term 97 (EK1100)^Term 102 (EL2809) A22^Channel 3^Output} *)
	STP.AUX20_AlumInService AT %QX48.0 : BOOL;	(*  ~ {LinkedWith:TIID^C6920 (EtherCAT)^ScadaRoom_KouplerUTP (EK1100)^ScadaRoom_KouplerFiber (EK1521)^ChemicalAndTertiary (EK1501)^Term 96 (EK1122)^Term 97 (EK1100)^Term 102 (EL2809) A22^Channel 4^Output} *)
	STP.AUX21_AlumInService AT %QX60.6 : BOOL;	(*  ~ {LinkedWith:TIID^C6920 (EtherCAT)^ScadaRoom_KouplerUTP (EK1100)^ScadaRoom_KouplerFiber (EK1521)^ChemicalAndTertiary (EK1501)^Term 96 (EK1122)^Term 97 (EK1100)^Term 102 (EL2809) A22^Channel 5^Output} *)
	STP.AUX22_AlumInService AT %QX48.3 : BOOL;	(*  ~ {LinkedWith:TIID^C6920 (EtherCAT)^ScadaRoom_KouplerUTP (EK1100)^ScadaRoom_KouplerFiber (EK1521)^ChemicalAndTertiary (EK1501)^Term 96 (EK1122)^Term 97 (EK1100)^Term 102 (EL2809) A22^Channel 6^Output} *)
	STP.AUX23_AlumInService AT %QX48.4 : BOOL;	(*  ~ {LinkedWith:TIID^C6920 (EtherCAT)^ScadaRoom_KouplerUTP (EK1100)^ScadaRoom_KouplerFiber (EK1521)^ChemicalAndTertiary (EK1501)^Term 96 (EK1122)^Term 97 (EK1100)^Term 102 (EL2809) A22^Channel 7^Output} *)
	STP.AUX24_CausticInService AT %QX48.5 : BOOL;	(*  ~ {LinkedWith:TIID^C6920 (EtherCAT)^ScadaRoom_KouplerUTP (EK1100)^ScadaRoom_KouplerFiber (EK1521)^ChemicalAndTertiary (EK1501)^Term 96 (EK1122)^Term 97 (EK1100)^Term 102 (EL2809) A22^Channel 8^Output} *)
	STP.AUX25_CausticInService AT %QX48.6 : BOOL;	(*  ~ {LinkedWith:TIID^C6920 (EtherCAT)^ScadaRoom_KouplerUTP (EK1100)^ScadaRoom_KouplerFiber (EK1521)^ChemicalAndTertiary (EK1501)^Term 96 (EK1122)^Term 97 (EK1100)^Term 102 (EL2809) A22^Channel 9^Output} *)
	STP.AUX26_SodiumInService AT %QX48.7 : BOOL;	(*  ~ {LinkedWith:TIID^C6920 (EtherCAT)^ScadaRoom_KouplerUTP (EK1100)^ScadaRoom_KouplerFiber (EK1521)^ChemicalAndTertiary (EK1501)^Term 96 (EK1122)^Term 97 (EK1100)^Term 102 (EL2809) A22^Channel 10^Output} *)
	STP.AUX27_SodiumInService AT %QX49.0 : BOOL;	(*  ~ {LinkedWith:TIID^C6920 (EtherCAT)^ScadaRoom_KouplerUTP (EK1100)^ScadaRoom_KouplerFiber (EK1521)^ChemicalAndTertiary (EK1501)^Term 96 (EK1122)^Term 97 (EK1100)^Term 102 (EL2809) A22^Channel 11^Output} *)
	STP.AUX28_SodiumInService AT %QX49.1 : BOOL;	(*  ~ {LinkedWith:TIID^C6920 (EtherCAT)^ScadaRoom_KouplerUTP (EK1100)^ScadaRoom_KouplerFiber (EK1521)^ChemicalAndTertiary (EK1501)^Term 96 (EK1122)^Term 97 (EK1100)^Term 102 (EL2809) A22^Channel 12^Output} *)
	STP.AUX33_LimeLOW AT %QX49.6 : BOOL;	(*  ~ {LinkedWith:TIID^C6920 (EtherCAT)^ScadaRoom_KouplerUTP (EK1100)^ScadaRoom_KouplerFiber (EK1521)^ChemicalAndTertiary (EK1501)^Term 96 (EK1122)^Term 97 (EK1100)^Term 103 (EL2809) A23^Channel 1^Output} *)
	STP.AUX34_LimeLOW AT %QX49.7 : BOOL;	(*  ~ {LinkedWith:TIID^C6920 (EtherCAT)^ScadaRoom_KouplerUTP (EK1100)^ScadaRoom_KouplerFiber (EK1521)^ChemicalAndTertiary (EK1501)^Term 96 (EK1122)^Term 97 (EK1100)^Term 103 (EL2809) A23^Channel 2^Output} *)
	STP.AUX35_LimeLOW AT %QX50.0 : BOOL;	(*  ~ {LinkedWith:TIID^C6920 (EtherCAT)^ScadaRoom_KouplerUTP (EK1100)^ScadaRoom_KouplerFiber (EK1521)^ChemicalAndTertiary (EK1501)^Term 96 (EK1122)^Term 97 (EK1100)^Term 103 (EL2809) A23^Channel 3^Output} *)
	STP.AUX36_AlumLOW AT %QX50.1 : BOOL;	(*  ~ {LinkedWith:TIID^C6920 (EtherCAT)^ScadaRoom_KouplerUTP (EK1100)^ScadaRoom_KouplerFiber (EK1521)^ChemicalAndTertiary (EK1501)^Term 96 (EK1122)^Term 97 (EK1100)^Term 103 (EL2809) A23^Channel 4^Output} *)
	STP.AUX37_AlumLOW AT %QX50.2 : BOOL;	(*  ~ {LinkedWith:TIID^C6920 (EtherCAT)^ScadaRoom_KouplerUTP (EK1100)^ScadaRoom_KouplerFiber (EK1521)^ChemicalAndTertiary (EK1501)^Term 96 (EK1122)^Term 97 (EK1100)^Term 103 (EL2809) A23^Channel 5^Output} *)
	STP.AUX38_AlumLOW AT %QX50.3 : BOOL;	(*  ~ {LinkedWith:TIID^C6920 (EtherCAT)^ScadaRoom_KouplerUTP (EK1100)^ScadaRoom_KouplerFiber (EK1521)^ChemicalAndTertiary (EK1501)^Term 96 (EK1122)^Term 97 (EK1100)^Term 103 (EL2809) A23^Channel 6^Output} *)
	STP.AUX39_AlumLOW AT %QX50.4 : BOOL;	(*  ~ {LinkedWith:TIID^C6920 (EtherCAT)^ScadaRoom_KouplerUTP (EK1100)^ScadaRoom_KouplerFiber (EK1521)^ChemicalAndTertiary (EK1501)^Term 96 (EK1122)^Term 97 (EK1100)^Term 103 (EL2809) A23^Channel 7^Output} *)
	STP.AUX40_CausticLOW AT %QX50.5 : BOOL;	(*  ~ {LinkedWith:TIID^C6920 (EtherCAT)^ScadaRoom_KouplerUTP (EK1100)^ScadaRoom_KouplerFiber (EK1521)^ChemicalAndTertiary (EK1501)^Term 96 (EK1122)^Term 97 (EK1100)^Term 103 (EL2809) A23^Channel 8^Output} *)
	STP.AUX41_CausticLOW AT %QX50.6 : BOOL;	(*  ~ {LinkedWith:TIID^C6920 (EtherCAT)^ScadaRoom_KouplerUTP (EK1100)^ScadaRoom_KouplerFiber (EK1521)^ChemicalAndTertiary (EK1501)^Term 96 (EK1122)^Term 97 (EK1100)^Term 103 (EL2809) A23^Channel 9^Output} *)
	STP.AUX42_SodiumLOW AT %QX50.7 : BOOL;	(*  ~ {LinkedWith:TIID^C6920 (EtherCAT)^ScadaRoom_KouplerUTP (EK1100)^ScadaRoom_KouplerFiber (EK1521)^ChemicalAndTertiary (EK1501)^Term 96 (EK1122)^Term 97 (EK1100)^Term 103 (EL2809) A23^Channel 10^Output} *)
	STP.AUX43_SodiumLOW AT %QX51.0 : BOOL;	(*  ~ {LinkedWith:TIID^C6920 (EtherCAT)^ScadaRoom_KouplerUTP (EK1100)^ScadaRoom_KouplerFiber (EK1521)^ChemicalAndTertiary (EK1501)^Term 96 (EK1122)^Term 97 (EK1100)^Term 103 (EL2809) A23^Channel 11^Output} *)
	STP.AUX44_SodiumLOW AT %QX51.1 : BOOL;	(*  ~ {LinkedWith:TIID^C6920 (EtherCAT)^ScadaRoom_KouplerUTP (EK1100)^ScadaRoom_KouplerFiber (EK1521)^ChemicalAndTertiary (EK1501)^Term 96 (EK1122)^Term 97 (EK1100)^Term 103 (EL2809) A23^Channel 12^Output} *)
	STP.FT300_EffluentFlowrateEntry_ScaledValue AT %IB526 : INT;	(*  ~ {LinkedWith:TIID^C6920 (EtherCAT)^ScadaRoom_KouplerUTP (EK1100)^ScadaRoom_KouplerFiber (EK1521)^ChemicalAndTertiary (EK1501)^Term 96 (EK1122)^Term 97 (EK1100)^Term 104 (EL3154) A24^AI Standard Channel 1^Value} *)
	STP.AT300_EffluentTurbidityEntry_ScaledValue AT %IB528 : INT;	(*  ~ {LinkedWith:TIID^C6920 (EtherCAT)^ScadaRoom_KouplerUTP (EK1100)^ScadaRoom_KouplerFiber (EK1521)^ChemicalAndTertiary (EK1501)^Term 96 (EK1122)^Term 97 (EK1100)^Term 104 (EL3154) A24^AI Standard Channel 2^Value} *)
	STP.PHT301_EffluentpHLevelEntry_ScaledValue AT %IB530 : INT;	(*  ~ {LinkedWith:TIID^C6920 (EtherCAT)^ScadaRoom_KouplerUTP (EK1100)^ScadaRoom_KouplerFiber (EK1521)^ChemicalAndTertiary (EK1501)^Term 96 (EK1122)^Term 97 (EK1100)^Term 104 (EL3154) A24^AI Standard Channel 3^Value} *)
	STP.FT301_TreatedEffluentFlowrateDischarge_ScaledValue AT %IB532 : INT;	(*  ~ {LinkedWith:TIID^C6920 (EtherCAT)^ScadaRoom_KouplerUTP (EK1100)^ScadaRoom_KouplerFiber (EK1521)^ChemicalAndTertiary (EK1501)^Term 96 (EK1122)^Term 97 (EK1100)^Term 105 (EL3154) A25^AI Standard Channel 1^Value} *)
	STP.AT302_TreatedEffluentTurbidityDischarge_ScaledValue AT %IB534 : INT;	(*  ~ {LinkedWith:TIID^C6920 (EtherCAT)^ScadaRoom_KouplerUTP (EK1100)^ScadaRoom_KouplerFiber (EK1521)^ChemicalAndTertiary (EK1501)^Term 96 (EK1122)^Term 97 (EK1100)^Term 105 (EL3154) A25^AI Standard Channel 2^Value} *)
	STP.PHT303_TreatedEffluentpHLevelDischarge_ScaledValue AT %IB536 : INT;	(*  ~ {LinkedWith:TIID^C6920 (EtherCAT)^ScadaRoom_KouplerUTP (EK1100)^ScadaRoom_KouplerFiber (EK1521)^ChemicalAndTertiary (EK1501)^Term 96 (EK1122)^Term 97 (EK1100)^Term 105 (EL3154) A25^AI Standard Channel 3^Value} *)
	STP.CL303_ResidualChlorineAnalyzer_ScaledValue AT %IB538 : INT;	(*  ~ {LinkedWith:TIID^C6920 (EtherCAT)^ScadaRoom_KouplerUTP (EK1100)^ScadaRoom_KouplerFiber (EK1521)^ChemicalAndTertiary (EK1501)^Term 96 (EK1122)^Term 97 (EK1100)^Term 106 (EL3154) A26^AI Standard Channel 1^Value} *)
	STP.CL304_FinalChlorineAnalyzer_ScaledValue AT %IB540 : INT;	(*  ~ {LinkedWith:TIID^C6920 (EtherCAT)^ScadaRoom_KouplerUTP (EK1100)^ScadaRoom_KouplerFiber (EK1521)^ChemicalAndTertiary (EK1501)^Term 96 (EK1122)^Term 97 (EK1100)^Term 106 (EL3154) A26^AI Standard Channel 2^Value} *)
	STP.ORP_DisinfectionTankAnalyzer_ScaledValue AT %IB542 : INT;	(*  ~ {LinkedWith:TIID^C6920 (EtherCAT)^ScadaRoom_KouplerUTP (EK1100)^ScadaRoom_KouplerFiber (EK1521)^ChemicalAndTertiary (EK1501)^Term 96 (EK1122)^Term 97 (EK1100)^Term 106 (EL3154) A26^AI Standard Channel 3^Value} *)
	STP.F500_FanStatus AT %IX456.6 : BOOL;	(*  ~ {LinkedWith:TIID^C6920 (EtherCAT)^ScadaRoom_KouplerUTP (EK1100)^ScadaRoom_KouplerFiber (EK1521)^SludgeThickening (EK1501)^Term 108 (EL1809) A2^Channel 1^Input} *)
	STP.D500_DoorPanelStatus AT %IX456.7 : BOOL;	(*  ~ {LinkedWith:TIID^C6920 (EtherCAT)^ScadaRoom_KouplerUTP (EK1100)^ScadaRoom_KouplerFiber (EK1521)^SludgeThickening (EK1501)^Term 108 (EL1809) A2^Channel 2^Input} *)
	STP.LSH501A_SludgeStorage AT %IX116.1 : BOOL;	(*  ~ {LinkedWith:TIID^C6920 (EtherCAT)^ScadaRoom_KouplerUTP (EK1100)^ScadaRoom_KouplerFiber (EK1521)^SludgeThickening (EK1501)^Term 108 (EL1809) A2^Channel 3^Input} *)
	STP.LSHH501A_SludgeStorage AT %IX116.2 : BOOL;	(*  ~ {LinkedWith:TIID^C6920 (EtherCAT)^ScadaRoom_KouplerUTP (EK1100)^ScadaRoom_KouplerFiber (EK1521)^SludgeThickening (EK1501)^Term 108 (EL1809) A2^Channel 4^Input} *)
	STP.LSL501A_SludgeStorage AT %IX116.3 : BOOL;	(*  ~ {LinkedWith:TIID^C6920 (EtherCAT)^ScadaRoom_KouplerUTP (EK1100)^ScadaRoom_KouplerFiber (EK1521)^SludgeThickening (EK1501)^Term 108 (EL1809) A2^Channel 5^Input} *)
	STP.LSH501B_SludgeStorage AT %IX116.4 : BOOL;	(*  ~ {LinkedWith:TIID^C6920 (EtherCAT)^ScadaRoom_KouplerUTP (EK1100)^ScadaRoom_KouplerFiber (EK1521)^SludgeThickening (EK1501)^Term 108 (EL1809) A2^Channel 6^Input} *)
	STP.LSHH501B_SludgeStorage AT %IX116.5 : BOOL;	(*  ~ {LinkedWith:TIID^C6920 (EtherCAT)^ScadaRoom_KouplerUTP (EK1100)^ScadaRoom_KouplerFiber (EK1521)^SludgeThickening (EK1501)^Term 108 (EL1809) A2^Channel 7^Input} *)
	STP.LSL501B_SludgeStorage AT %IX116.6 : BOOL;	(*  ~ {LinkedWith:TIID^C6920 (EtherCAT)^ScadaRoom_KouplerUTP (EK1100)^ScadaRoom_KouplerFiber (EK1521)^SludgeThickening (EK1501)^Term 108 (EL1809) A2^Channel 8^Input} *)
	STP.LSH620_FiltrateSumpLevel AT %IX116.7 : BOOL;	(*  ~ {LinkedWith:TIID^C6920 (EtherCAT)^ScadaRoom_KouplerUTP (EK1100)^ScadaRoom_KouplerFiber (EK1521)^SludgeThickening (EK1501)^Term 108 (EL1809) A2^Channel 9^Input} *)
	STP.LSL620_FiltrateSumpLevel AT %IX117.0 : BOOL;	(*  ~ {LinkedWith:TIID^C6920 (EtherCAT)^ScadaRoom_KouplerUTP (EK1100)^ScadaRoom_KouplerFiber (EK1521)^SludgeThickening (EK1501)^Term 108 (EL1809) A2^Channel 10^Input} *)
	STP.LSHPU501_PolymerTankLevel AT %IX117.1 : BOOL;	(*  ~ {LinkedWith:TIID^C6920 (EtherCAT)^ScadaRoom_KouplerUTP (EK1100)^ScadaRoom_KouplerFiber (EK1521)^SludgeThickening (EK1501)^Term 108 (EL1809) A2^Channel 12^Input} *)
	STP.LSLPU501_PolymerTankLevel AT %IX117.2 : BOOL;	(*  ~ {LinkedWith:TIID^C6920 (EtherCAT)^ScadaRoom_KouplerUTP (EK1100)^ScadaRoom_KouplerFiber (EK1521)^SludgeThickening (EK1501)^Term 108 (EL1809) A2^Channel 11^Input} *)
	STP.PSL505A_PressureSWWaterLine AT %IX117.3 : BOOL;	(*  ~ {LinkedWith:TIID^C6920 (EtherCAT)^ScadaRoom_KouplerUTP (EK1100)^ScadaRoom_KouplerFiber (EK1521)^SludgeThickening (EK1501)^Term 108 (EL1809) A2^Channel 13^Input} *)
	STP.PSL505B_PressureSWWaterLine2 AT %IX117.4 : BOOL;	(*  ~ {LinkedWith:TIID^C6920 (EtherCAT)^ScadaRoom_KouplerUTP (EK1100)^ScadaRoom_KouplerFiber (EK1521)^SludgeThickening (EK1501)^Term 108 (EL1809) A2^Channel 14^Input} *)
	STP.P501A_SludgeFeedPump_RunStat AT %IX117.5 : BOOL;	(*  ~ {LinkedWith:TIID^C6920 (EtherCAT)^ScadaRoom_KouplerUTP (EK1100)^ScadaRoom_KouplerFiber (EK1521)^SludgeThickening (EK1501)^Term 109 (EL1809) A3^Channel 1^Input} *)
	STP.P501B_SludgeFeedPump_RunStat AT %IX117.6 : BOOL;	(*  ~ {LinkedWith:TIID^C6920 (EtherCAT)^ScadaRoom_KouplerUTP (EK1100)^ScadaRoom_KouplerFiber (EK1521)^SludgeThickening (EK1501)^Term 109 (EL1809) A3^Channel 2^Input} *)
	STP.P501C_SludgeFeedPump_RunStat AT %IX117.7 : BOOL;	(*  ~ {LinkedWith:TIID^C6920 (EtherCAT)^ScadaRoom_KouplerUTP (EK1100)^ScadaRoom_KouplerFiber (EK1521)^SludgeThickening (EK1501)^Term 109 (EL1809) A3^Channel 3^Input} *)
	STP.B501A_Blower_RunStat AT %IX118.0 : BOOL;	(*  ~ {LinkedWith:TIID^C6920 (EtherCAT)^ScadaRoom_KouplerUTP (EK1100)^ScadaRoom_KouplerFiber (EK1521)^SludgeThickening (EK1501)^Term 109 (EL1809) A3^Channel 4^Input} *)
	STP.B501B_Blower_RunStat AT %IX118.1 : BOOL;	(*  ~ {LinkedWith:TIID^C6920 (EtherCAT)^ScadaRoom_KouplerUTP (EK1100)^ScadaRoom_KouplerFiber (EK1521)^SludgeThickening (EK1501)^Term 109 (EL1809) A3^Channel 5^Input} *)
	STP.B501C_Blower_RunStat AT %IX118.2 : BOOL;	(*  ~ {LinkedWith:TIID^C6920 (EtherCAT)^ScadaRoom_KouplerUTP (EK1100)^ScadaRoom_KouplerFiber (EK1521)^SludgeThickening (EK1501)^Term 109 (EL1809) A3^Channel 6^Input} *)
	STP.M502A_Floculator_RunStat AT %IX118.3 : BOOL;	(*  ~ {LinkedWith:TIID^C6920 (EtherCAT)^ScadaRoom_KouplerUTP (EK1100)^ScadaRoom_KouplerFiber (EK1521)^SludgeThickening (EK1501)^Term 109 (EL1809) A3^Channel 7^Input} *)
	STP.M502B_Floculator_RunStat AT %IX118.4 : BOOL;	(*  ~ {LinkedWith:TIID^C6920 (EtherCAT)^ScadaRoom_KouplerUTP (EK1100)^ScadaRoom_KouplerFiber (EK1521)^SludgeThickening (EK1501)^Term 109 (EL1809) A3^Channel 8^Input} *)
	STP.P602A_FiltratePump_RunStat AT %IX118.5 : BOOL;	(*  ~ {LinkedWith:TIID^C6920 (EtherCAT)^ScadaRoom_KouplerUTP (EK1100)^ScadaRoom_KouplerFiber (EK1521)^SludgeThickening (EK1501)^Term 109 (EL1809) A3^Channel 9^Input} *)
	STP.P602B_FiltratePump_RunStat AT %IX118.6 : BOOL;	(*  ~ {LinkedWith:TIID^C6920 (EtherCAT)^ScadaRoom_KouplerUTP (EK1100)^ScadaRoom_KouplerFiber (EK1521)^SludgeThickening (EK1501)^Term 109 (EL1809) A3^Channel 10^Input} *)
	STP.XV505A_SolenoidValveLine_OpenStat AT %IX118.7 : BOOL;	(*  ~ {LinkedWith:TIID^C6920 (EtherCAT)^ScadaRoom_KouplerUTP (EK1100)^ScadaRoom_KouplerFiber (EK1521)^SludgeThickening (EK1501)^Term 109 (EL1809) A3^Channel 11^Input} *)
	STP.XV505B_SolenoidValveLine_OpenStat AT %IX119.0 : BOOL;	(*  ~ {LinkedWith:TIID^C6920 (EtherCAT)^ScadaRoom_KouplerUTP (EK1100)^ScadaRoom_KouplerFiber (EK1521)^SludgeThickening (EK1501)^Term 109 (EL1809) A3^Channel 12^Input} *)
	STP.XVPU502_DiagpharmAirValve_OpenStat AT %IX119.1 : BOOL;	(*  ~ {LinkedWith:TIID^C6920 (EtherCAT)^ScadaRoom_KouplerUTP (EK1100)^ScadaRoom_KouplerFiber (EK1521)^SludgeThickening (EK1501)^Term 109 (EL1809) A3^Channel 13^Input} *)
	STP.XV505A_SolenoidValveLine_CloseStat AT %IX119.2 : BOOL;	(*  ~ {LinkedWith:TIID^C6920 (EtherCAT)^ScadaRoom_KouplerUTP (EK1100)^ScadaRoom_KouplerFiber (EK1521)^SludgeThickening (EK1501)^Term 109 (EL1809) A3^Channel 14^Input} *)
	STP.XV505B_SolenoidValveLine_CloseStat AT %IX119.3 : BOOL;	(*  ~ {LinkedWith:TIID^C6920 (EtherCAT)^ScadaRoom_KouplerUTP (EK1100)^ScadaRoom_KouplerFiber (EK1521)^SludgeThickening (EK1501)^Term 109 (EL1809) A3^Channel 15^Input} *)
	STP.XVPU502_DiagpharmAirValve_CloseStat AT %IX119.4 : BOOL;	(*  ~ {LinkedWith:TIID^C6920 (EtherCAT)^ScadaRoom_KouplerUTP (EK1100)^ScadaRoom_KouplerFiber (EK1521)^SludgeThickening (EK1501)^Term 109 (EL1809) A3^Channel 16^Input} *)
	STP.D503A_DrumThickener_RunStat AT %IX262.4 : BOOL;	(*  ~ {LinkedWith:TIID^C6920 (EtherCAT)^ScadaRoom_KouplerUTP (EK1100)^ScadaRoom_KouplerFiber (EK1521)^SludgeThickening (EK1501)^Term 110 (EL1809) A4^Channel 1^Input} *)
	STP.D503B_DrumThickener_RunStat AT %IX262.5 : BOOL;	(*  ~ {LinkedWith:TIID^C6920 (EtherCAT)^ScadaRoom_KouplerUTP (EK1100)^ScadaRoom_KouplerFiber (EK1521)^SludgeThickening (EK1501)^Term 110 (EL1809) A4^Channel 2^Input} *)
	STP.P505A_BackwashWaterPump_RunStat AT %IX262.6 : BOOL;	(*  ~ {LinkedWith:TIID^C6920 (EtherCAT)^ScadaRoom_KouplerUTP (EK1100)^ScadaRoom_KouplerFiber (EK1521)^SludgeThickening (EK1501)^Term 110 (EL1809) A4^Channel 3^Input} *)
	STP.P505B_BackwashWaterPump_RunStat AT %IX262.7 : BOOL;	(*  ~ {LinkedWith:TIID^C6920 (EtherCAT)^ScadaRoom_KouplerUTP (EK1100)^ScadaRoom_KouplerFiber (EK1521)^SludgeThickening (EK1501)^Term 110 (EL1809) A4^Channel 4^Input} *)
	STP.P505C_BackwashWaterPump_RunStat AT %IX263.0 : BOOL;	(*  ~ {LinkedWith:TIID^C6920 (EtherCAT)^ScadaRoom_KouplerUTP (EK1100)^ScadaRoom_KouplerFiber (EK1521)^SludgeThickening (EK1501)^Term 110 (EL1809) A4^Channel 5^Input} *)
	STP.XV501A_AirBlowerValve_OpenStat AT %IX120.2 : BOOL;	(*  ~ {LinkedWith:TIID^C6920 (EtherCAT)^ScadaRoom_KouplerUTP (EK1100)^ScadaRoom_KouplerFiber (EK1521)^SludgeThickening (EK1501)^Term 110 (EL1809) A4^Channel 6^Input} *)
	STP.XV501A_AirBlowerValve_CloseStat AT %IX120.3 : BOOL;	(*  ~ {LinkedWith:TIID^C6920 (EtherCAT)^ScadaRoom_KouplerUTP (EK1100)^ScadaRoom_KouplerFiber (EK1521)^SludgeThickening (EK1501)^Term 110 (EL1809) A4^Channel 7^Input} *)
	STP.XV501B_AirBlowerValve_OpenStat AT %IX120.4 : BOOL;	(*  ~ {LinkedWith:TIID^C6920 (EtherCAT)^ScadaRoom_KouplerUTP (EK1100)^ScadaRoom_KouplerFiber (EK1521)^SludgeThickening (EK1501)^Term 110 (EL1809) A4^Channel 8^Input} *)
	STP.XV501B_AirBlowerValve_CloseStat AT %IX120.5 : BOOL;	(*  ~ {LinkedWith:TIID^C6920 (EtherCAT)^ScadaRoom_KouplerUTP (EK1100)^ScadaRoom_KouplerFiber (EK1521)^SludgeThickening (EK1501)^Term 110 (EL1809) A4^Channel 9^Input} *)
	STP.XVPU501A_PolymerValve_OpenStat AT %IX120.6 : BOOL;	(*  ~ {LinkedWith:TIID^C6920 (EtherCAT)^ScadaRoom_KouplerUTP (EK1100)^ScadaRoom_KouplerFiber (EK1521)^SludgeThickening (EK1501)^Term 110 (EL1809) A4^Channel 10^Input} *)
	STP.XVPU501A_PolymerValve_CloseStat AT %IX120.7 : BOOL;	(*  ~ {LinkedWith:TIID^C6920 (EtherCAT)^ScadaRoom_KouplerUTP (EK1100)^ScadaRoom_KouplerFiber (EK1521)^SludgeThickening (EK1501)^Term 110 (EL1809) A4^Channel 11^Input} *)
	STP.XVPU501B_PolymerValve_OpenStat AT %IX121.0 : BOOL;	(*  ~ {LinkedWith:TIID^C6920 (EtherCAT)^ScadaRoom_KouplerUTP (EK1100)^ScadaRoom_KouplerFiber (EK1521)^SludgeThickening (EK1501)^Term 110 (EL1809) A4^Channel 12^Input} *)
	STP.XVPU501B_PolymerValve_CloseStat AT %IX328.0 : BOOL;	(*  ~ {LinkedWith:TIID^C6920 (EtherCAT)^ScadaRoom_KouplerUTP (EK1100)^ScadaRoom_KouplerFiber (EK1521)^SludgeThickening (EK1501)^Term 110 (EL1809) A4^Channel 13^Input} *)
	STP.M503_PolymerStirrer_RunStat AT %IX263.1 : BOOL;	(*  ~ {LinkedWith:TIID^C6920 (EtherCAT)^ScadaRoom_KouplerUTP (EK1100)^ScadaRoom_KouplerFiber (EK1521)^SludgeThickening (EK1501)^Term 110 (EL1809) A4^Channel 14^Input} *)
	STP.XVW501A_WaterValve_OpenStat AT %IX292.0 : BOOL;	(*  ~ {LinkedWith:TIID^C6920 (EtherCAT)^ScadaRoom_KouplerUTP (EK1100)^ScadaRoom_KouplerFiber (EK1521)^SludgeThickening (EK1501)^Term 110 (EL1809) A4^Channel 15^Input} *)
	STP.XVW501A_WaterValve_CloseStat AT %IX292.1 : BOOL;	(*  ~ {LinkedWith:TIID^C6920 (EtherCAT)^ScadaRoom_KouplerUTP (EK1100)^ScadaRoom_KouplerFiber (EK1521)^SludgeThickening (EK1501)^Term 110 (EL1809) A4^Channel 16^Input} *)
	STP.B501A_Blower_OverloadStat AT %IX121.3 : BOOL;	(*  ~ {LinkedWith:TIID^C6920 (EtherCAT)^ScadaRoom_KouplerUTP (EK1100)^ScadaRoom_KouplerFiber (EK1521)^SludgeThickening (EK1501)^Term 111 (EL1809) A5^Channel 1^Input} *)
	STP.B501A_Blower_IncompleteStat AT %IX121.4 : BOOL;	(*  ~ {LinkedWith:TIID^C6920 (EtherCAT)^ScadaRoom_KouplerUTP (EK1100)^ScadaRoom_KouplerFiber (EK1521)^SludgeThickening (EK1501)^Term 111 (EL1809) A5^Channel 2^Input} *)
	STP.B501B_Blower_OverloadStat AT %IX121.5 : BOOL;	(*  ~ {LinkedWith:TIID^C6920 (EtherCAT)^ScadaRoom_KouplerUTP (EK1100)^ScadaRoom_KouplerFiber (EK1521)^SludgeThickening (EK1501)^Term 111 (EL1809) A5^Channel 3^Input} *)
	STP.B501B_Blower_IncompleteStat AT %IX121.6 : BOOL;	(*  ~ {LinkedWith:TIID^C6920 (EtherCAT)^ScadaRoom_KouplerUTP (EK1100)^ScadaRoom_KouplerFiber (EK1521)^SludgeThickening (EK1501)^Term 111 (EL1809) A5^Channel 4^Input} *)
	STP.B501C_Blower_OverloadStat AT %IX121.7 : BOOL;	(*  ~ {LinkedWith:TIID^C6920 (EtherCAT)^ScadaRoom_KouplerUTP (EK1100)^ScadaRoom_KouplerFiber (EK1521)^SludgeThickening (EK1501)^Term 111 (EL1809) A5^Channel 5^Input} *)
	STP.B501C_Blower_IncompleteStat AT %IX122.0 : BOOL;	(*  ~ {LinkedWith:TIID^C6920 (EtherCAT)^ScadaRoom_KouplerUTP (EK1100)^ScadaRoom_KouplerFiber (EK1521)^SludgeThickening (EK1501)^Term 111 (EL1809) A5^Channel 6^Input} *)
	STP.P501A_SludgeFeedPump_OverloadStat AT %IX122.1 : BOOL;	(*  ~ {LinkedWith:TIID^C6920 (EtherCAT)^ScadaRoom_KouplerUTP (EK1100)^ScadaRoom_KouplerFiber (EK1521)^SludgeThickening (EK1501)^Term 111 (EL1809) A5^Channel 7^Input} *)
	STP.P501A_SludgeFeedPump_IncompleteStat AT %IX122.2 : BOOL;	(*  ~ {LinkedWith:TIID^C6920 (EtherCAT)^ScadaRoom_KouplerUTP (EK1100)^ScadaRoom_KouplerFiber (EK1521)^SludgeThickening (EK1501)^Term 111 (EL1809) A5^Channel 8^Input} *)
	STP.P501B_SludgeFeedPump_OverloadStat AT %IX122.3 : BOOL;	(*  ~ {LinkedWith:TIID^C6920 (EtherCAT)^ScadaRoom_KouplerUTP (EK1100)^ScadaRoom_KouplerFiber (EK1521)^SludgeThickening (EK1501)^Term 111 (EL1809) A5^Channel 9^Input} *)
	STP.P501B_SludgeFeedPump_IncompleteStat AT %IX122.4 : BOOL;	(*  ~ {LinkedWith:TIID^C6920 (EtherCAT)^ScadaRoom_KouplerUTP (EK1100)^ScadaRoom_KouplerFiber (EK1521)^SludgeThickening (EK1501)^Term 111 (EL1809) A5^Channel 10^Input} *)
	STP.P501C_SludgeFeedPumpOverloadStat AT %IX122.5 : BOOL;	(*  ~ {LinkedWith:TIID^C6920 (EtherCAT)^ScadaRoom_KouplerUTP (EK1100)^ScadaRoom_KouplerFiber (EK1521)^SludgeThickening (EK1501)^Term 111 (EL1809) A5^Channel 11^Input} *)
	STP.P501C_SludgeFeedPump_IncompleteStat AT %IX122.6 : BOOL;	(*  ~ {LinkedWith:TIID^C6920 (EtherCAT)^ScadaRoom_KouplerUTP (EK1100)^ScadaRoom_KouplerFiber (EK1521)^SludgeThickening (EK1501)^Term 111 (EL1809) A5^Channel 12^Input} *)
	STP.P602A_FiltratePump_TripStat AT %IX263.2 : BOOL;	(*  ~ {LinkedWith:TIID^C6920 (EtherCAT)^ScadaRoom_KouplerUTP (EK1100)^ScadaRoom_KouplerFiber (EK1521)^SludgeThickening (EK1501)^Term 111 (EL1809) A5^Channel 13^Input} *)
	STP.P602B_FiltratePump_TripStat AT %IX263.3 : BOOL;	(*  ~ {LinkedWith:TIID^C6920 (EtherCAT)^ScadaRoom_KouplerUTP (EK1100)^ScadaRoom_KouplerFiber (EK1521)^SludgeThickening (EK1501)^Term 111 (EL1809) A5^Channel 14^Input} *)
	STP.M502A_Floculator_OverloadStat AT %IX123.1 : BOOL;	(*  ~ {LinkedWith:TIID^C6920 (EtherCAT)^ScadaRoom_KouplerUTP (EK1100)^ScadaRoom_KouplerFiber (EK1521)^SludgeThickening (EK1501)^Term 112 (EL1809) A6^Channel 1^Input} *)
	STP.M502B_Floculator_OverloadStat AT %IX123.2 : BOOL;	(*  ~ {LinkedWith:TIID^C6920 (EtherCAT)^ScadaRoom_KouplerUTP (EK1100)^ScadaRoom_KouplerFiber (EK1521)^SludgeThickening (EK1501)^Term 112 (EL1809) A6^Channel 2^Input} *)
	STP.D503A_DrumThickener_OverloadStat AT %IX123.3 : BOOL;	(*  ~ {LinkedWith:TIID^C6920 (EtherCAT)^ScadaRoom_KouplerUTP (EK1100)^ScadaRoom_KouplerFiber (EK1521)^SludgeThickening (EK1501)^Term 112 (EL1809) A6^Channel 3^Input} *)
	STP.D503B_DrumThickener_OverloadStat AT %IX123.4 : BOOL;	(*  ~ {LinkedWith:TIID^C6920 (EtherCAT)^ScadaRoom_KouplerUTP (EK1100)^ScadaRoom_KouplerFiber (EK1521)^SludgeThickening (EK1501)^Term 112 (EL1809) A6^Channel 4^Input} *)
	STP.P505A_BackwashWaterPump_OverloadStat AT %IX123.5 : BOOL;	(*  ~ {LinkedWith:TIID^C6920 (EtherCAT)^ScadaRoom_KouplerUTP (EK1100)^ScadaRoom_KouplerFiber (EK1521)^SludgeThickening (EK1501)^Term 112 (EL1809) A6^Channel 5^Input} *)
	STP.P505B_BackwashWaterPump_OverloadStat AT %IX123.7 : BOOL;	(*  ~ {LinkedWith:TIID^C6920 (EtherCAT)^ScadaRoom_KouplerUTP (EK1100)^ScadaRoom_KouplerFiber (EK1521)^SludgeThickening (EK1501)^Term 112 (EL1809) A6^Channel 7^Input} *)
	STP.P505C_BackwashWaterPump_OverloadStat AT %IX124.1 : BOOL;	(*  ~ {LinkedWith:TIID^C6920 (EtherCAT)^ScadaRoom_KouplerUTP (EK1100)^ScadaRoom_KouplerFiber (EK1521)^SludgeThickening (EK1501)^Term 112 (EL1809) A6^Channel 9^Input} *)
	STP.M503_PolymerStirrer_OverloadStat AT %IX124.3 : BOOL;	(*  ~ {LinkedWith:TIID^C6920 (EtherCAT)^ScadaRoom_KouplerUTP (EK1100)^ScadaRoom_KouplerFiber (EK1521)^SludgeThickening (EK1501)^Term 112 (EL1809) A6^Channel 11^Input} *)
	STP.P501A_SludgeFeedPump_LocalRemoteStat AT %IX263.4 : BOOL;	(*  ~ {LinkedWith:TIID^C6920 (EtherCAT)^ScadaRoom_KouplerUTP (EK1100)^ScadaRoom_KouplerFiber (EK1521)^SludgeThickening (EK1501)^Term 113 (EL1809) A7^Channel 1^Input} *)
	STP.P501B_SludgeFeedPump_LocalRemoteStat AT %IX263.5 : BOOL;	(*  ~ {LinkedWith:TIID^C6920 (EtherCAT)^ScadaRoom_KouplerUTP (EK1100)^ScadaRoom_KouplerFiber (EK1521)^SludgeThickening (EK1501)^Term 113 (EL1809) A7^Channel 2^Input} *)
	STP.P501C_SludgeFeedPump_LocalRemoteStat AT %IX263.6 : BOOL;	(*  ~ {LinkedWith:TIID^C6920 (EtherCAT)^ScadaRoom_KouplerUTP (EK1100)^ScadaRoom_KouplerFiber (EK1521)^SludgeThickening (EK1501)^Term 113 (EL1809) A7^Channel 3^Input} *)
	STP.B501A_Blower_LocalRemoteStat AT %IX263.7 : BOOL;	(*  ~ {LinkedWith:TIID^C6920 (EtherCAT)^ScadaRoom_KouplerUTP (EK1100)^ScadaRoom_KouplerFiber (EK1521)^SludgeThickening (EK1501)^Term 113 (EL1809) A7^Channel 4^Input} *)
	STP.B501B_Blower_LocalRemoteStat AT %IX264.0 : BOOL;	(*  ~ {LinkedWith:TIID^C6920 (EtherCAT)^ScadaRoom_KouplerUTP (EK1100)^ScadaRoom_KouplerFiber (EK1521)^SludgeThickening (EK1501)^Term 113 (EL1809) A7^Channel 5^Input} *)
	STP.B501C_Blower_LocalRemoteStat AT %IX264.1 : BOOL;	(*  ~ {LinkedWith:TIID^C6920 (EtherCAT)^ScadaRoom_KouplerUTP (EK1100)^ScadaRoom_KouplerFiber (EK1521)^SludgeThickening (EK1501)^Term 113 (EL1809) A7^Channel 6^Input} *)
	STP.M502A_Floculator_LocalRemoteStat AT %IX264.2 : BOOL;	(*  ~ {LinkedWith:TIID^C6920 (EtherCAT)^ScadaRoom_KouplerUTP (EK1100)^ScadaRoom_KouplerFiber (EK1521)^SludgeThickening (EK1501)^Term 113 (EL1809) A7^Channel 7^Input} *)
	STP.M502B_Floculator_LocalRemoteStat AT %IX264.3 : BOOL;	(*  ~ {LinkedWith:TIID^C6920 (EtherCAT)^ScadaRoom_KouplerUTP (EK1100)^ScadaRoom_KouplerFiber (EK1521)^SludgeThickening (EK1501)^Term 113 (EL1809) A7^Channel 8^Input} *)
	STP.D503A_DrumThickener_LocalRemoteStat AT %IX264.4 : BOOL;	(*  ~ {LinkedWith:TIID^C6920 (EtherCAT)^ScadaRoom_KouplerUTP (EK1100)^ScadaRoom_KouplerFiber (EK1521)^SludgeThickening (EK1501)^Term 113 (EL1809) A7^Channel 9^Input} *)
	STP.D503B_DrumThickener_LocalRemoteStat AT %IX264.5 : BOOL;	(*  ~ {LinkedWith:TIID^C6920 (EtherCAT)^ScadaRoom_KouplerUTP (EK1100)^ScadaRoom_KouplerFiber (EK1521)^SludgeThickening (EK1501)^Term 113 (EL1809) A7^Channel 10^Input} *)
	STP.P505A_BackwashWaterPump_LocalRemoteStat AT %IX264.6 : BOOL;	(*  ~ {LinkedWith:TIID^C6920 (EtherCAT)^ScadaRoom_KouplerUTP (EK1100)^ScadaRoom_KouplerFiber (EK1521)^SludgeThickening (EK1501)^Term 113 (EL1809) A7^Channel 11^Input} *)
	STP.P505B_BackwashWaterPump_LocalRemoteStat AT %IX264.7 : BOOL;	(*  ~ {LinkedWith:TIID^C6920 (EtherCAT)^ScadaRoom_KouplerUTP (EK1100)^ScadaRoom_KouplerFiber (EK1521)^SludgeThickening (EK1501)^Term 113 (EL1809) A7^Channel 12^Input} *)
	STP.P505C_BackwashWaterPump_LocalRemoteStat AT %IX265.0 : BOOL;	(*  ~ {LinkedWith:TIID^C6920 (EtherCAT)^ScadaRoom_KouplerUTP (EK1100)^ScadaRoom_KouplerFiber (EK1521)^SludgeThickening (EK1501)^Term 113 (EL1809) A7^Channel 13^Input} *)
	STP.P602A_FiltratePump_LocalRemoteStat AT %IX122.7 : BOOL;	(*  ~ {LinkedWith:TIID^C6920 (EtherCAT)^ScadaRoom_KouplerUTP (EK1100)^ScadaRoom_KouplerFiber (EK1521)^SludgeThickening (EK1501)^Term 113 (EL1809) A7^Channel 14^Input} *)
	STP.P602B_FiltratePump_LocalRemoteStat AT %IX123.0 : BOOL;	(*  ~ {LinkedWith:TIID^C6920 (EtherCAT)^ScadaRoom_KouplerUTP (EK1100)^ScadaRoom_KouplerFiber (EK1521)^SludgeThickening (EK1501)^Term 113 (EL1809) A7^Channel 15^Input} *)
	STP.M503_PolymerStirrer_LocalRemoteStat AT %IX265.1 : BOOL;	(*  ~ {LinkedWith:TIID^C6920 (EtherCAT)^ScadaRoom_KouplerUTP (EK1100)^ScadaRoom_KouplerFiber (EK1521)^SludgeThickening (EK1501)^Term 113 (EL1809) A7^Channel 16^Input} *)
	STP.P501A_SludgeFeedPump_EStopStat AT %IX126.4 : BOOL;	(*  ~ {LinkedWith:TIID^C6920 (EtherCAT)^ScadaRoom_KouplerUTP (EK1100)^ScadaRoom_KouplerFiber (EK1521)^SludgeThickening (EK1501)^Term 114 (EL1809) A8^Channel 1^Input} *)
	STP.P501B_SludgeFeedPump_EStopStat AT %IX126.5 : BOOL;	(*  ~ {LinkedWith:TIID^C6920 (EtherCAT)^ScadaRoom_KouplerUTP (EK1100)^ScadaRoom_KouplerFiber (EK1521)^SludgeThickening (EK1501)^Term 114 (EL1809) A8^Channel 2^Input} *)
	STP.P501C_SludgeFeedPump_EStopStat AT %IX126.6 : BOOL;	(*  ~ {LinkedWith:TIID^C6920 (EtherCAT)^ScadaRoom_KouplerUTP (EK1100)^ScadaRoom_KouplerFiber (EK1521)^SludgeThickening (EK1501)^Term 114 (EL1809) A8^Channel 3^Input} *)
	STP.B501A_Blower_EStopStat AT %IX126.7 : BOOL;	(*  ~ {LinkedWith:TIID^C6920 (EtherCAT)^ScadaRoom_KouplerUTP (EK1100)^ScadaRoom_KouplerFiber (EK1521)^SludgeThickening (EK1501)^Term 114 (EL1809) A8^Channel 4^Input} *)
	STP.B501B_Blower_EStopStat AT %IX127.0 : BOOL;	(*  ~ {LinkedWith:TIID^C6920 (EtherCAT)^ScadaRoom_KouplerUTP (EK1100)^ScadaRoom_KouplerFiber (EK1521)^SludgeThickening (EK1501)^Term 114 (EL1809) A8^Channel 5^Input} *)
	STP.B501C_Blower_EStopStat AT %IX127.1 : BOOL;	(*  ~ {LinkedWith:TIID^C6920 (EtherCAT)^ScadaRoom_KouplerUTP (EK1100)^ScadaRoom_KouplerFiber (EK1521)^SludgeThickening (EK1501)^Term 114 (EL1809) A8^Channel 6^Input} *)
	STP.M502A_Floculator_EStopStat AT %IX127.2 : BOOL;	(*  ~ {LinkedWith:TIID^C6920 (EtherCAT)^ScadaRoom_KouplerUTP (EK1100)^ScadaRoom_KouplerFiber (EK1521)^SludgeThickening (EK1501)^Term 114 (EL1809) A8^Channel 7^Input} *)
	STP.M502B_Floculator_EStopStat AT %IX127.3 : BOOL;	(*  ~ {LinkedWith:TIID^C6920 (EtherCAT)^ScadaRoom_KouplerUTP (EK1100)^ScadaRoom_KouplerFiber (EK1521)^SludgeThickening (EK1501)^Term 114 (EL1809) A8^Channel 8^Input} *)
	STP.D503A_DrumThickener_EStopStat AT %IX127.4 : BOOL;	(*  ~ {LinkedWith:TIID^C6920 (EtherCAT)^ScadaRoom_KouplerUTP (EK1100)^ScadaRoom_KouplerFiber (EK1521)^SludgeThickening (EK1501)^Term 114 (EL1809) A8^Channel 9^Input} *)
	STP.D503B_DrumThickener_EStopStat AT %IX127.5 : BOOL;	(*  ~ {LinkedWith:TIID^C6920 (EtherCAT)^ScadaRoom_KouplerUTP (EK1100)^ScadaRoom_KouplerFiber (EK1521)^SludgeThickening (EK1501)^Term 114 (EL1809) A8^Channel 10^Input} *)
	STP.P505A_BackwashWaterPump_EStopStat AT %IX127.6 : BOOL;	(*  ~ {LinkedWith:TIID^C6920 (EtherCAT)^ScadaRoom_KouplerUTP (EK1100)^ScadaRoom_KouplerFiber (EK1521)^SludgeThickening (EK1501)^Term 114 (EL1809) A8^Channel 11^Input} *)
	STP.P505B_BackwashWaterPump_EStopStat AT %IX127.7 : BOOL;	(*  ~ {LinkedWith:TIID^C6920 (EtherCAT)^ScadaRoom_KouplerUTP (EK1100)^ScadaRoom_KouplerFiber (EK1521)^SludgeThickening (EK1501)^Term 114 (EL1809) A8^Channel 12^Input} *)
	STP.P505C_BackwashWaterPump_EStopStat AT %IX128.0 : BOOL;	(*  ~ {LinkedWith:TIID^C6920 (EtherCAT)^ScadaRoom_KouplerUTP (EK1100)^ScadaRoom_KouplerFiber (EK1521)^SludgeThickening (EK1501)^Term 114 (EL1809) A8^Channel 13^Input} *)
	STP.P602A_FiltratePump_EStopStat AT %IX128.1 : BOOL;	(*  ~ {LinkedWith:TIID^C6920 (EtherCAT)^ScadaRoom_KouplerUTP (EK1100)^ScadaRoom_KouplerFiber (EK1521)^SludgeThickening (EK1501)^Term 114 (EL1809) A8^Channel 14^Input} *)
	STP.P602B_FiltratePump_EStopStat AT %IX128.2 : BOOL;	(*  ~ {LinkedWith:TIID^C6920 (EtherCAT)^ScadaRoom_KouplerUTP (EK1100)^ScadaRoom_KouplerFiber (EK1521)^SludgeThickening (EK1501)^Term 114 (EL1809) A8^Channel 15^Input} *)
	STP.M503_PolymerStirrer_EStopStat AT %IX128.3 : BOOL;	(*  ~ {LinkedWith:TIID^C6920 (EtherCAT)^ScadaRoom_KouplerUTP (EK1100)^ScadaRoom_KouplerFiber (EK1521)^SludgeThickening (EK1501)^Term 114 (EL1809) A8^Channel 16^Input} *)
	STP.VE801B_SuctionFan_OnOffStat AT %IX265.2 : BOOL;	(*  ~ {LinkedWith:TIID^C6920 (EtherCAT)^ScadaRoom_KouplerUTP (EK1100)^ScadaRoom_KouplerFiber (EK1521)^SludgeThickening (EK1501)^Term 115 (EL1809) A9^Channel 1^Input} *)
	STP.P802B_CirculationPump_OnOffStat AT %IX265.3 : BOOL;	(*  ~ {LinkedWith:TIID^C6920 (EtherCAT)^ScadaRoom_KouplerUTP (EK1100)^ScadaRoom_KouplerFiber (EK1521)^SludgeThickening (EK1501)^Term 115 (EL1809) A9^Channel 2^Input} *)
	STP.P803B_CirculationPump_OnOffStat AT %IX265.4 : BOOL;	(*  ~ {LinkedWith:TIID^C6920 (EtherCAT)^ScadaRoom_KouplerUTP (EK1100)^ScadaRoom_KouplerFiber (EK1521)^SludgeThickening (EK1501)^Term 115 (EL1809) A9^Channel 3^Input} *)
	STP.P804B_CirculationPump_OnOffStat AT %IX265.5 : BOOL;	(*  ~ {LinkedWith:TIID^C6920 (EtherCAT)^ScadaRoom_KouplerUTP (EK1100)^ScadaRoom_KouplerFiber (EK1521)^SludgeThickening (EK1501)^Term 115 (EL1809) A9^Channel 4^Input} *)
	STP.P805B1_H2S04Pump_OnOffStat AT %IX265.6 : BOOL;	(*  ~ {LinkedWith:TIID^C6920 (EtherCAT)^ScadaRoom_KouplerUTP (EK1100)^ScadaRoom_KouplerFiber (EK1521)^SludgeThickening (EK1501)^Term 115 (EL1809) A9^Channel 5^Input} *)
	STP.P805B2_H2S04Pump_OnOffStat AT %IX265.7 : BOOL;	(*  ~ {LinkedWith:TIID^C6920 (EtherCAT)^ScadaRoom_KouplerUTP (EK1100)^ScadaRoom_KouplerFiber (EK1521)^SludgeThickening (EK1501)^Term 115 (EL1809) A9^Channel 6^Input} *)
	STP.P806B1_NAOHPump_OnOffStat AT %IX266.0 : BOOL;	(*  ~ {LinkedWith:TIID^C6920 (EtherCAT)^ScadaRoom_KouplerUTP (EK1100)^ScadaRoom_KouplerFiber (EK1521)^SludgeThickening (EK1501)^Term 115 (EL1809) A9^Channel 7^Input} *)
	STP.P806B2_NAOHPump_OnOffStat AT %IX266.1 : BOOL;	(*  ~ {LinkedWith:TIID^C6920 (EtherCAT)^ScadaRoom_KouplerUTP (EK1100)^ScadaRoom_KouplerFiber (EK1521)^SludgeThickening (EK1501)^Term 115 (EL1809) A9^Channel 8^Input} *)
	STP.P807B1_NAOCLPump_OnOffStat AT %IX266.2 : BOOL;	(*  ~ {LinkedWith:TIID^C6920 (EtherCAT)^ScadaRoom_KouplerUTP (EK1100)^ScadaRoom_KouplerFiber (EK1521)^SludgeThickening (EK1501)^Term 115 (EL1809) A9^Channel 9^Input} *)
	STP.P807B2_NAOCLPump_OnOffStat AT %IX266.3 : BOOL;	(*  ~ {LinkedWith:TIID^C6920 (EtherCAT)^ScadaRoom_KouplerUTP (EK1100)^ScadaRoom_KouplerFiber (EK1521)^SludgeThickening (EK1501)^Term 115 (EL1809) A9^Channel 10^Input} *)
	STP.VE801B_SuctionFan_OverloadStat AT %IX266.4 : BOOL;	(*  ~ {LinkedWith:TIID^C6920 (EtherCAT)^ScadaRoom_KouplerUTP (EK1100)^ScadaRoom_KouplerFiber (EK1521)^SludgeThickening (EK1501)^Term 115 (EL1809) A9^Channel 11^Input} *)
	STP.P802B_CirculationPump_OverloadStat AT %IX266.5 : BOOL;	(*  ~ {LinkedWith:TIID^C6920 (EtherCAT)^ScadaRoom_KouplerUTP (EK1100)^ScadaRoom_KouplerFiber (EK1521)^SludgeThickening (EK1501)^Term 115 (EL1809) A9^Channel 12^Input} *)
	STP.P803B_CirculationPump_OverloadStat AT %IX266.6 : BOOL;	(*  ~ {LinkedWith:TIID^C6920 (EtherCAT)^ScadaRoom_KouplerUTP (EK1100)^ScadaRoom_KouplerFiber (EK1521)^SludgeThickening (EK1501)^Term 115 (EL1809) A9^Channel 13^Input} *)
	STP.P804B_CirculationPump_OverloadStat AT %IX266.7 : BOOL;	(*  ~ {LinkedWith:TIID^C6920 (EtherCAT)^ScadaRoom_KouplerUTP (EK1100)^ScadaRoom_KouplerFiber (EK1521)^SludgeThickening (EK1501)^Term 115 (EL1809) A9^Channel 14^Input} *)
	STP.P805B1_H2S04Pump_OverloadStat AT %IX267.0 : BOOL;	(*  ~ {LinkedWith:TIID^C6920 (EtherCAT)^ScadaRoom_KouplerUTP (EK1100)^ScadaRoom_KouplerFiber (EK1521)^SludgeThickening (EK1501)^Term 115 (EL1809) A9^Channel 15^Input} *)
	STP.P805B2_H2S04Pump_OverloadStat AT %IX267.1 : BOOL;	(*  ~ {LinkedWith:TIID^C6920 (EtherCAT)^ScadaRoom_KouplerUTP (EK1100)^ScadaRoom_KouplerFiber (EK1521)^SludgeThickening (EK1501)^Term 115 (EL1809) A9^Channel 16^Input} *)
	STP.P806B1_NAOHPump_OverloadStat AT %IX267.2 : BOOL;	(*  ~ {LinkedWith:TIID^C6920 (EtherCAT)^ScadaRoom_KouplerUTP (EK1100)^ScadaRoom_KouplerFiber (EK1521)^SludgeThickening (EK1501)^Term 116 (EL1809) A10^Channel 1^Input} *)
	STP.P806B2_NAOHPump_OverloadStat AT %IX267.3 : BOOL;	(*  ~ {LinkedWith:TIID^C6920 (EtherCAT)^ScadaRoom_KouplerUTP (EK1100)^ScadaRoom_KouplerFiber (EK1521)^SludgeThickening (EK1501)^Term 116 (EL1809) A10^Channel 2^Input} *)
	STP.P807B1_NAOCLPump_OverloadStat AT %IX267.4 : BOOL;	(*  ~ {LinkedWith:TIID^C6920 (EtherCAT)^ScadaRoom_KouplerUTP (EK1100)^ScadaRoom_KouplerFiber (EK1521)^SludgeThickening (EK1501)^Term 116 (EL1809) A10^Channel 3^Input} *)
	STP.P807B2_NAOCLPump_OverloadStat AT %IX267.5 : BOOL;	(*  ~ {LinkedWith:TIID^C6920 (EtherCAT)^ScadaRoom_KouplerUTP (EK1100)^ScadaRoom_KouplerFiber (EK1521)^SludgeThickening (EK1501)^Term 116 (EL1809) A10^Channel 4^Input} *)
	STP.VE801B_Suction_EStopStat AT %IX267.6 : BOOL;	(*  ~ {LinkedWith:TIID^C6920 (EtherCAT)^ScadaRoom_KouplerUTP (EK1100)^ScadaRoom_KouplerFiber (EK1521)^SludgeThickening (EK1501)^Term 116 (EL1809) A10^Channel 5^Input} *)
	STP.P802B_CirculationPump_EStopStat AT %IX267.7 : BOOL;	(*  ~ {LinkedWith:TIID^C6920 (EtherCAT)^ScadaRoom_KouplerUTP (EK1100)^ScadaRoom_KouplerFiber (EK1521)^SludgeThickening (EK1501)^Term 116 (EL1809) A10^Channel 6^Input} *)
	STP.P803B_CirculationPump_EStopStat AT %IX268.0 : BOOL;	(*  ~ {LinkedWith:TIID^C6920 (EtherCAT)^ScadaRoom_KouplerUTP (EK1100)^ScadaRoom_KouplerFiber (EK1521)^SludgeThickening (EK1501)^Term 116 (EL1809) A10^Channel 7^Input} *)
	STP.P804B_CirculationPump_EStopStat AT %IX268.1 : BOOL;	(*  ~ {LinkedWith:TIID^C6920 (EtherCAT)^ScadaRoom_KouplerUTP (EK1100)^ScadaRoom_KouplerFiber (EK1521)^SludgeThickening (EK1501)^Term 116 (EL1809) A10^Channel 8^Input} *)
	STP.P805B1_H2S04Pump_EStopStat AT %IX268.2 : BOOL;	(*  ~ {LinkedWith:TIID^C6920 (EtherCAT)^ScadaRoom_KouplerUTP (EK1100)^ScadaRoom_KouplerFiber (EK1521)^SludgeThickening (EK1501)^Term 116 (EL1809) A10^Channel 9^Input} *)
	STP.P805B2_H2S04Pump_EStopStat AT %IX268.3 : BOOL;	(*  ~ {LinkedWith:TIID^C6920 (EtherCAT)^ScadaRoom_KouplerUTP (EK1100)^ScadaRoom_KouplerFiber (EK1521)^SludgeThickening (EK1501)^Term 116 (EL1809) A10^Channel 10^Input} *)
	STP.P806B1_NAOHPump_EStopStat AT %IX268.4 : BOOL;	(*  ~ {LinkedWith:TIID^C6920 (EtherCAT)^ScadaRoom_KouplerUTP (EK1100)^ScadaRoom_KouplerFiber (EK1521)^SludgeThickening (EK1501)^Term 116 (EL1809) A10^Channel 11^Input} *)
	STP.P806B2_NAOHPump_EstopStat AT %IX268.5 : BOOL;	(*  ~ {LinkedWith:TIID^C6920 (EtherCAT)^ScadaRoom_KouplerUTP (EK1100)^ScadaRoom_KouplerFiber (EK1521)^SludgeThickening (EK1501)^Term 116 (EL1809) A10^Channel 12^Input} *)
	STP.P807B1_NAOCLPump_EStopStat AT %IX268.6 : BOOL;	(*  ~ {LinkedWith:TIID^C6920 (EtherCAT)^ScadaRoom_KouplerUTP (EK1100)^ScadaRoom_KouplerFiber (EK1521)^SludgeThickening (EK1501)^Term 116 (EL1809) A10^Channel 13^Input} *)
	STP.P807B2_NAOCLPump_EStopStat AT %IX268.7 : BOOL;	(*  ~ {LinkedWith:TIID^C6920 (EtherCAT)^ScadaRoom_KouplerUTP (EK1100)^ScadaRoom_KouplerFiber (EK1521)^SludgeThickening (EK1501)^Term 116 (EL1809) A10^Channel 14^Input} *)
	STP.LSH600_SludgePitSensor_ScaledValue AT %IB544 : INT;	(*  ~ {LinkedWith:TIID^C6920 (EtherCAT)^ScadaRoom_KouplerUTP (EK1100)^ScadaRoom_KouplerFiber (EK1521)^SludgeThickening (EK1501)^Term 117 (EL3154) A11^AI Standard Channel 1^Value} *)
	STP.XVPU502_DiagpharmAirValve_OpenCmd AT %QX60.7 : BOOL;	(*  ~ {LinkedWith:TIID^C6920 (EtherCAT)^ScadaRoom_KouplerUTP (EK1100)^ScadaRoom_KouplerFiber (EK1521)^SludgeThickening (EK1501)^Term 118 (EL2809) A12^Channel 1^Output} *)
	STP.M502A_Floculator_RunCmd AT %QX100.0 : BOOL;	(*  ~ {LinkedWith:TIID^C6920 (EtherCAT)^ScadaRoom_KouplerUTP (EK1100)^ScadaRoom_KouplerFiber (EK1521)^SludgeThickening (EK1501)^Term 118 (EL2809) A12^Channel 2^Output} *)
	STP.M502B_Floculator_RunCmd AT %QX100.1 : BOOL;	(*  ~ {LinkedWith:TIID^C6920 (EtherCAT)^ScadaRoom_KouplerUTP (EK1100)^ScadaRoom_KouplerFiber (EK1521)^SludgeThickening (EK1501)^Term 118 (EL2809) A12^Channel 3^Output} *)
	STP.D503A_DrumThickener_RunCmd AT %QX96.2 : BOOL;	(*  ~ {LinkedWith:TIID^C6920 (EtherCAT)^ScadaRoom_KouplerUTP (EK1100)^ScadaRoom_KouplerFiber (EK1521)^SludgeThickening (EK1501)^Term 118 (EL2809) A12^Channel 4^Output} *)
	STP.D503B_DrumThickener_RunCmd AT %QX100.2 : BOOL;	(*  ~ {LinkedWith:TIID^C6920 (EtherCAT)^ScadaRoom_KouplerUTP (EK1100)^ScadaRoom_KouplerFiber (EK1521)^SludgeThickening (EK1501)^Term 118 (EL2809) A12^Channel 5^Output} *)
	STP.P602A_FiltratePump_RunCmd AT %QX61.6 : BOOL;	(*  ~ {LinkedWith:TIID^C6920 (EtherCAT)^ScadaRoom_KouplerUTP (EK1100)^ScadaRoom_KouplerFiber (EK1521)^SludgeThickening (EK1501)^Term 118 (EL2809) A12^Channel 8^Output} *)
	STP.P602B_FiltratePump_RunCmd AT %QX61.7 : BOOL;	(*  ~ {LinkedWith:TIID^C6920 (EtherCAT)^ScadaRoom_KouplerUTP (EK1100)^ScadaRoom_KouplerFiber (EK1521)^SludgeThickening (EK1501)^Term 118 (EL2809) A12^Channel 9^Output} *)
	STP.XVPU501A_PolymerValve_OpenCloseCmd AT %QX104.0 : BOOL;	(*  ~ {LinkedWith:TIID^C6920 (EtherCAT)^ScadaRoom_KouplerUTP (EK1100)^ScadaRoom_KouplerFiber (EK1521)^SludgeThickening (EK1501)^Term 118 (EL2809) A12^Channel 10^Output} *)
	STP.XVPU501B_PolymerValve_OpenCloseCmd AT %QX104.1 : BOOL;	(*  ~ {LinkedWith:TIID^C6920 (EtherCAT)^ScadaRoom_KouplerUTP (EK1100)^ScadaRoom_KouplerFiber (EK1521)^SludgeThickening (EK1501)^Term 118 (EL2809) A12^Channel 11^Output} *)
	STP.XV505A_SolenoidValveLine_OpenCmd AT %QX62.4 : BOOL;	(*  ~ {LinkedWith:TIID^C6920 (EtherCAT)^ScadaRoom_KouplerUTP (EK1100)^ScadaRoom_KouplerFiber (EK1521)^SludgeThickening (EK1501)^Term 118 (EL2809) A12^Channel 14^Output} *)
	STP.XV505B_SolenoidValveLine_CloseCmd AT %QX62.5 : BOOL;	(*  ~ {LinkedWith:TIID^C6920 (EtherCAT)^ScadaRoom_KouplerUTP (EK1100)^ScadaRoom_KouplerFiber (EK1521)^SludgeThickening (EK1501)^Term 118 (EL2809) A12^Channel 15^Output} *)
	STP.XVW501A_WaterValve_OpenCmd AT %QX73.3 : BOOL;	(*  ~ {LinkedWith:TIID^C6920 (EtherCAT)^ScadaRoom_KouplerUTP (EK1100)^ScadaRoom_KouplerFiber (EK1521)^SludgeThickening (EK1501)^Term 118 (EL2809) A12^Channel 16^Output} *)
	STP.B501A_Blower_RunCmd AT %QX62.6 : BOOL;	(*  ~ {LinkedWith:TIID^C6920 (EtherCAT)^ScadaRoom_KouplerUTP (EK1100)^ScadaRoom_KouplerFiber (EK1521)^SludgeThickening (EK1501)^Term 119 (EL2809) A13^Channel 1^Output} *)
	STP.B501B_Blower_RunCmd AT %QX62.7 : BOOL;	(*  ~ {LinkedWith:TIID^C6920 (EtherCAT)^ScadaRoom_KouplerUTP (EK1100)^ScadaRoom_KouplerFiber (EK1521)^SludgeThickening (EK1501)^Term 119 (EL2809) A13^Channel 2^Output} *)
	STP.B501C_Blower_RunCmd AT %QX63.0 : BOOL;	(*  ~ {LinkedWith:TIID^C6920 (EtherCAT)^ScadaRoom_KouplerUTP (EK1100)^ScadaRoom_KouplerFiber (EK1521)^SludgeThickening (EK1501)^Term 119 (EL2809) A13^Channel 3^Output} *)
	STP.P501A_SludgeFeedPump_RunCmd AT %QX63.1 : BOOL;	(*  ~ {LinkedWith:TIID^C6920 (EtherCAT)^ScadaRoom_KouplerUTP (EK1100)^ScadaRoom_KouplerFiber (EK1521)^SludgeThickening (EK1501)^Term 119 (EL2809) A13^Channel 4^Output} *)
	STP.P501B_SludgeFeedPump_RunCmd AT %QX63.2 : BOOL;	(*  ~ {LinkedWith:TIID^C6920 (EtherCAT)^ScadaRoom_KouplerUTP (EK1100)^ScadaRoom_KouplerFiber (EK1521)^SludgeThickening (EK1501)^Term 119 (EL2809) A13^Channel 5^Output} *)
	STP.P501C_SludgeFeedPump_RunCmd AT %QX63.3 : BOOL;	(*  ~ {LinkedWith:TIID^C6920 (EtherCAT)^ScadaRoom_KouplerUTP (EK1100)^ScadaRoom_KouplerFiber (EK1521)^SludgeThickening (EK1501)^Term 119 (EL2809) A13^Channel 6^Output} *)
	STP.P505A_BackwashWaterPump_RunCmd AT %QX63.4 : BOOL;	(*  ~ {LinkedWith:TIID^C6920 (EtherCAT)^ScadaRoom_KouplerUTP (EK1100)^ScadaRoom_KouplerFiber (EK1521)^SludgeThickening (EK1501)^Term 119 (EL2809) A13^Channel 7^Output} *)
	STP.P505B_BackwashWaterPump_RunCmd AT %QX63.5 : BOOL;	(*  ~ {LinkedWith:TIID^C6920 (EtherCAT)^ScadaRoom_KouplerUTP (EK1100)^ScadaRoom_KouplerFiber (EK1521)^SludgeThickening (EK1501)^Term 119 (EL2809) A13^Channel 8^Output} *)
	STP.P505C_BackwashWaterPump_RunCmd AT %QX63.6 : BOOL;	(*  ~ {LinkedWith:TIID^C6920 (EtherCAT)^ScadaRoom_KouplerUTP (EK1100)^ScadaRoom_KouplerFiber (EK1521)^SludgeThickening (EK1501)^Term 119 (EL2809) A13^Channel 9^Output} *)
	STP.XV501A_AirBlowerValve_OpenCmd AT %QX63.7 : BOOL;	(*  ~ {LinkedWith:TIID^C6920 (EtherCAT)^ScadaRoom_KouplerUTP (EK1100)^ScadaRoom_KouplerFiber (EK1521)^SludgeThickening (EK1501)^Term 119 (EL2809) A13^Channel 10^Output} *)
	STP.XV501B_AirBlowerValve_OpenCmd AT %QX64.0 : BOOL;	(*  ~ {LinkedWith:TIID^C6920 (EtherCAT)^ScadaRoom_KouplerUTP (EK1100)^ScadaRoom_KouplerFiber (EK1521)^SludgeThickening (EK1501)^Term 119 (EL2809) A13^Channel 11^Output} *)
	STP.XV501A_AirBlowerValve_CloseCmd AT %QX64.1 : BOOL;	(*  ~ {LinkedWith:TIID^C6920 (EtherCAT)^ScadaRoom_KouplerUTP (EK1100)^ScadaRoom_KouplerFiber (EK1521)^SludgeThickening (EK1501)^Term 119 (EL2809) A13^Channel 12^Output} *)
	STP.XV501B_AirBlowerValve_CloseCmd AT %QX64.2 : BOOL;	(*  ~ {LinkedWith:TIID^C6920 (EtherCAT)^ScadaRoom_KouplerUTP (EK1100)^ScadaRoom_KouplerFiber (EK1521)^SludgeThickening (EK1501)^Term 119 (EL2809) A13^Channel 13^Output} *)
	STP.M503_PolymerStirrer_FwdCmd AT %QX64.3 : BOOL;	(*  ~ {LinkedWith:TIID^C6920 (EtherCAT)^ScadaRoom_KouplerUTP (EK1100)^ScadaRoom_KouplerFiber (EK1521)^SludgeThickening (EK1501)^Term 119 (EL2809) A13^Channel 14^Output} *)
	STP.M503_PolymerStirrer_RvsCmd AT %QX64.4 : BOOL;	(*  ~ {LinkedWith:TIID^C6920 (EtherCAT)^ScadaRoom_KouplerUTP (EK1100)^ScadaRoom_KouplerFiber (EK1521)^SludgeThickening (EK1501)^Term 119 (EL2809) A13^Channel 15^Output} *)
	STP.AUX510_SludgeStorageHigh AT %QX73.4 : BOOL;	(*  ~ {LinkedWith:TIID^C6920 (EtherCAT)^ScadaRoom_KouplerUTP (EK1100)^ScadaRoom_KouplerFiber (EK1521)^SludgeThickening (EK1501)^Term 120 (EL2809) A14^Channel 1^Output} *)
	STP.AUX511_ReuseWaterStorageLow AT %QX64.7 : BOOL;	(*  ~ {LinkedWith:TIID^C6920 (EtherCAT)^ScadaRoom_KouplerUTP (EK1100)^ScadaRoom_KouplerFiber (EK1521)^SludgeThickening (EK1501)^Term 120 (EL2809) A14^Channel 2^Output} *)
	STP.AUX512_FiltrateSumpHigh AT %QX73.5 : BOOL;	(*  ~ {LinkedWith:TIID^C6920 (EtherCAT)^ScadaRoom_KouplerUTP (EK1100)^ScadaRoom_KouplerFiber (EK1521)^SludgeThickening (EK1501)^Term 120 (EL2809) A14^Channel 3^Output} *)
	STP.AUX513_SludgePitHigh AT %QX73.6 : BOOL;	(*  ~ {LinkedWith:TIID^C6920 (EtherCAT)^ScadaRoom_KouplerUTP (EK1100)^ScadaRoom_KouplerFiber (EK1521)^SludgeThickening (EK1501)^Term 120 (EL2809) A14^Channel 4^Output} *)
	STP.AUX514_PolymerLevelLow AT %QX65.2 : BOOL;	(*  ~ {LinkedWith:TIID^C6920 (EtherCAT)^ScadaRoom_KouplerUTP (EK1100)^ScadaRoom_KouplerFiber (EK1521)^SludgeThickening (EK1501)^Term 120 (EL2809) A14^Channel 5^Output} *)
	STP.AUX701_CommonAlarm AT %QX73.7 : BOOL;	(*  ~ {LinkedWith:TIID^C6920 (EtherCAT)^ScadaRoom_KouplerUTP (EK1100)^ScadaRoom_KouplerFiber (EK1521)^SludgeThickening (EK1501)^Term 120 (EL2809) A14^Channel 6^Output} *)
	STP.AUX702_PLCRunStat AT %QX74.0 : BOOL;	(*  ~ {LinkedWith:TIID^C6920 (EtherCAT)^ScadaRoom_KouplerUTP (EK1100)^ScadaRoom_KouplerFiber (EK1521)^SludgeThickening (EK1501)^Term 120 (EL2809) A14^Channel 7^Output} *)
	STP.LSL309A_WaterLevelTank AT %IX269.0 : BOOL;	(*  ~ {LinkedWith:TIID^C6920 (EtherCAT)^ScadaRoom_KouplerUTP (EK1100)^ScadaRoom_KouplerFiber (EK1521)^Reused (EK1501)^Term 122 (EL1809) A2^Channel 1^Input} *)
	STP.LSL309B_WaterLevelTank AT %IX269.1 : BOOL;	(*  ~ {LinkedWith:TIID^C6920 (EtherCAT)^ScadaRoom_KouplerUTP (EK1100)^ScadaRoom_KouplerFiber (EK1521)^Reused (EK1501)^Term 122 (EL1809) A2^Channel 2^Input} *)
	STP.LSH405_VacuumChestLevel AT %IX132.4 : BOOL;	(*  ~ {LinkedWith:TIID^C6920 (EtherCAT)^ScadaRoom_KouplerUTP (EK1100)^ScadaRoom_KouplerFiber (EK1521)^Reused (EK1501)^Term 122 (EL1809) A2^Channel 3^Input} *)
	STP.F400_FanStatus AT %IX457.0 : BOOL;	(*  ~ {LinkedWith:TIID^C6920 (EtherCAT)^ScadaRoom_KouplerUTP (EK1100)^ScadaRoom_KouplerFiber (EK1521)^Reused (EK1501)^Term 122 (EL1809) A2^Channel 4^Input} *)
	STP.D400_DoorPanelStatus AT %IX457.1 : BOOL;	(*  ~ {LinkedWith:TIID^C6920 (EtherCAT)^ScadaRoom_KouplerUTP (EK1100)^ScadaRoom_KouplerFiber (EK1521)^Reused (EK1501)^Term 122 (EL1809) A2^Channel 5^Input} *)
	STP.FSL101_FreshWaterActivationStatus AT %IX132.7 : BOOL;	(*  ~ {LinkedWith:TIID^C6920 (EtherCAT)^ScadaRoom_KouplerUTP (EK1100)^ScadaRoom_KouplerFiber (EK1521)^Reused (EK1501)^Term 122 (EL1809) A2^Channel 6^Input} *)
	STP.PSL412_PressureSwitch AT %IX133.0 : BOOL;	(*  ~ {LinkedWith:TIID^C6920 (EtherCAT)^ScadaRoom_KouplerUTP (EK1100)^ScadaRoom_KouplerFiber (EK1521)^Reused (EK1501)^Term 122 (EL1809) A2^Channel 7^Input} *)
	STP.PG413_LowPressureGauge AT %IX133.1 : BOOL;	(*  ~ {LinkedWith:TIID^C6920 (EtherCAT)^ScadaRoom_KouplerUTP (EK1100)^ScadaRoom_KouplerFiber (EK1521)^Reused (EK1501)^Term 122 (EL1809) A2^Channel 8^Input} *)
	STP.PG414_HighPressureGauge AT %IX133.2 : BOOL;	(*  ~ {LinkedWith:TIID^C6920 (EtherCAT)^ScadaRoom_KouplerUTP (EK1100)^ScadaRoom_KouplerFiber (EK1521)^Reused (EK1501)^Term 122 (EL1809) A2^Channel 9^Input} *)
	STP.XV401_SolenoidValve_OpenStat AT %IX133.3 : BOOL;	(*  ~ {LinkedWith:TIID^C6920 (EtherCAT)^ScadaRoom_KouplerUTP (EK1100)^ScadaRoom_KouplerFiber (EK1521)^Reused (EK1501)^Term 122 (EL1809) A2^Channel 10^Input} *)
	STP.XV401_SolenoidValve_CloseStat AT %IX133.4 : BOOL;	(*  ~ {LinkedWith:TIID^C6920 (EtherCAT)^ScadaRoom_KouplerUTP (EK1100)^ScadaRoom_KouplerFiber (EK1521)^Reused (EK1501)^Term 122 (EL1809) A2^Channel 11^Input} *)
	STP.P401A_LeadPumpA_OverloadStat AT %IX133.5 : BOOL;	(*  ~ {LinkedWith:TIID^C6920 (EtherCAT)^ScadaRoom_KouplerUTP (EK1100)^ScadaRoom_KouplerFiber (EK1521)^Reused (EK1501)^Term 123 (EL1809) A3^Channel 1^Input} *)
	STP.P401A_LeadPumpA_IncompleteStat AT %IX133.6 : BOOL;	(*  ~ {LinkedWith:TIID^C6920 (EtherCAT)^ScadaRoom_KouplerUTP (EK1100)^ScadaRoom_KouplerFiber (EK1521)^Reused (EK1501)^Term 123 (EL1809) A3^Channel 2^Input} *)
	STP.P401B_LeadPumpB_OverloadStat AT %IX133.7 : BOOL;	(*  ~ {LinkedWith:TIID^C6920 (EtherCAT)^ScadaRoom_KouplerUTP (EK1100)^ScadaRoom_KouplerFiber (EK1521)^Reused (EK1501)^Term 123 (EL1809) A3^Channel 3^Input} *)
	STP.P401B_LeadPumpB_IncompleteStat AT %IX134.0 : BOOL;	(*  ~ {LinkedWith:TIID^C6920 (EtherCAT)^ScadaRoom_KouplerUTP (EK1100)^ScadaRoom_KouplerFiber (EK1521)^Reused (EK1501)^Term 123 (EL1809) A3^Channel 4^Input} *)
	STP.P401C_LeadPumpC_OverloadStat AT %IX134.1 : BOOL;	(*  ~ {LinkedWith:TIID^C6920 (EtherCAT)^ScadaRoom_KouplerUTP (EK1100)^ScadaRoom_KouplerFiber (EK1521)^Reused (EK1501)^Term 123 (EL1809) A3^Channel 5^Input} *)
	STP.P401C_LeadPumpC_IncompleteStat AT %IX134.2 : BOOL;	(*  ~ {LinkedWith:TIID^C6920 (EtherCAT)^ScadaRoom_KouplerUTP (EK1100)^ScadaRoom_KouplerFiber (EK1521)^Reused (EK1501)^Term 123 (EL1809) A3^Channel 6^Input} *)
	STP.P401D_LeadPumpD_OverloadStat AT %IX134.3 : BOOL;	(*  ~ {LinkedWith:TIID^C6920 (EtherCAT)^ScadaRoom_KouplerUTP (EK1100)^ScadaRoom_KouplerFiber (EK1521)^Reused (EK1501)^Term 123 (EL1809) A3^Channel 7^Input} *)
	STP.P401D_LeadPumpD_IncompleteStat AT %IX134.4 : BOOL;	(*  ~ {LinkedWith:TIID^C6920 (EtherCAT)^ScadaRoom_KouplerUTP (EK1100)^ScadaRoom_KouplerFiber (EK1521)^Reused (EK1501)^Term 123 (EL1809) A3^Channel 8^Input} *)
	STP.P402A_JockeyPumpA_OverloadStat AT %IX134.5 : BOOL;	(*  ~ {LinkedWith:TIID^C6920 (EtherCAT)^ScadaRoom_KouplerUTP (EK1100)^ScadaRoom_KouplerFiber (EK1521)^Reused (EK1501)^Term 123 (EL1809) A3^Channel 9^Input} *)
	STP.P402A_JockeyPumpA_IncompleteStat AT %IX134.6 : BOOL;	(*  ~ {LinkedWith:TIID^C6920 (EtherCAT)^ScadaRoom_KouplerUTP (EK1100)^ScadaRoom_KouplerFiber (EK1521)^Reused (EK1501)^Term 123 (EL1809) A3^Channel 10^Input} *)
	STP.P402B_JockeyPumpB_OverloadStat AT %IX134.7 : BOOL;	(*  ~ {LinkedWith:TIID^C6920 (EtherCAT)^ScadaRoom_KouplerUTP (EK1100)^ScadaRoom_KouplerFiber (EK1521)^Reused (EK1501)^Term 123 (EL1809) A3^Channel 11^Input} *)
	STP.P402B_JockeyPumpB_IncompleteStat AT %IX135.0 : BOOL;	(*  ~ {LinkedWith:TIID^C6920 (EtherCAT)^ScadaRoom_KouplerUTP (EK1100)^ScadaRoom_KouplerFiber (EK1521)^Reused (EK1501)^Term 123 (EL1809) A3^Channel 12^Input} *)
	STP.P403A_VacuumPumpA_OverloadStat AT %IX135.1 : BOOL;	(*  ~ {LinkedWith:TIID^C6920 (EtherCAT)^ScadaRoom_KouplerUTP (EK1100)^ScadaRoom_KouplerFiber (EK1521)^Reused (EK1501)^Term 123 (EL1809) A3^Channel 13^Input} *)
	STP.P403B_VacuumPumpB_OverloadStat AT %IX135.3 : BOOL;	(*  ~ {LinkedWith:TIID^C6920 (EtherCAT)^ScadaRoom_KouplerUTP (EK1100)^ScadaRoom_KouplerFiber (EK1521)^Reused (EK1501)^Term 123 (EL1809) A3^Channel 15^Input} *)
	STP.P401A_LeadPumpA_LocalRemoteStat AT %IX135.5 : BOOL;	(*  ~ {LinkedWith:TIID^C6920 (EtherCAT)^ScadaRoom_KouplerUTP (EK1100)^ScadaRoom_KouplerFiber (EK1521)^Reused (EK1501)^Term 124 (EL1809) A4^Channel 1^Input} *)
	STP.P401B_LeadPumpB_LocalRemoteStat AT %IX135.6 : BOOL;	(*  ~ {LinkedWith:TIID^C6920 (EtherCAT)^ScadaRoom_KouplerUTP (EK1100)^ScadaRoom_KouplerFiber (EK1521)^Reused (EK1501)^Term 124 (EL1809) A4^Channel 2^Input} *)
	STP.P401C_LeadPumpC_LocalRemoteStat AT %IX135.7 : BOOL;	(*  ~ {LinkedWith:TIID^C6920 (EtherCAT)^ScadaRoom_KouplerUTP (EK1100)^ScadaRoom_KouplerFiber (EK1521)^Reused (EK1501)^Term 124 (EL1809) A4^Channel 3^Input} *)
	STP.P401D_LeadPumpD_LocalRemoteStat AT %IX136.0 : BOOL;	(*  ~ {LinkedWith:TIID^C6920 (EtherCAT)^ScadaRoom_KouplerUTP (EK1100)^ScadaRoom_KouplerFiber (EK1521)^Reused (EK1501)^Term 124 (EL1809) A4^Channel 4^Input} *)
	STP.P402A_JockeyPumpA_LocalRemoteStat AT %IX136.1 : BOOL;	(*  ~ {LinkedWith:TIID^C6920 (EtherCAT)^ScadaRoom_KouplerUTP (EK1100)^ScadaRoom_KouplerFiber (EK1521)^Reused (EK1501)^Term 124 (EL1809) A4^Channel 5^Input} *)
	STP.P402B_JockeyPumpB_LocalRemoteStat AT %IX136.2 : BOOL;	(*  ~ {LinkedWith:TIID^C6920 (EtherCAT)^ScadaRoom_KouplerUTP (EK1100)^ScadaRoom_KouplerFiber (EK1521)^Reused (EK1501)^Term 124 (EL1809) A4^Channel 6^Input} *)
	STP.P403A_VacuumPumpA_LocalRemoteStat AT %IX136.3 : BOOL;	(*  ~ {LinkedWith:TIID^C6920 (EtherCAT)^ScadaRoom_KouplerUTP (EK1100)^ScadaRoom_KouplerFiber (EK1521)^Reused (EK1501)^Term 124 (EL1809) A4^Channel 7^Input} *)
	STP.P403B_VacuumPumpB_LocalRemoteStat AT %IX136.4 : BOOL;	(*  ~ {LinkedWith:TIID^C6920 (EtherCAT)^ScadaRoom_KouplerUTP (EK1100)^ScadaRoom_KouplerFiber (EK1521)^Reused (EK1501)^Term 124 (EL1809) A4^Channel 8^Input} *)
	STP.P401A_LeadPumpA_OnOffStat AT %IX136.5 : BOOL;	(*  ~ {LinkedWith:TIID^C6920 (EtherCAT)^ScadaRoom_KouplerUTP (EK1100)^ScadaRoom_KouplerFiber (EK1521)^Reused (EK1501)^Term 124 (EL1809) A4^Channel 9^Input} *)
	STP.P401B_LeadPumpB_OnOffStat AT %IX136.6 : BOOL;	(*  ~ {LinkedWith:TIID^C6920 (EtherCAT)^ScadaRoom_KouplerUTP (EK1100)^ScadaRoom_KouplerFiber (EK1521)^Reused (EK1501)^Term 124 (EL1809) A4^Channel 10^Input} *)
	STP.P401C_LeadPumpC_OnOffStat AT %IX136.7 : BOOL;	(*  ~ {LinkedWith:TIID^C6920 (EtherCAT)^ScadaRoom_KouplerUTP (EK1100)^ScadaRoom_KouplerFiber (EK1521)^Reused (EK1501)^Term 124 (EL1809) A4^Channel 11^Input} *)
	STP.P401D_LeadPumpD_OnOffStat AT %IX137.0 : BOOL;	(*  ~ {LinkedWith:TIID^C6920 (EtherCAT)^ScadaRoom_KouplerUTP (EK1100)^ScadaRoom_KouplerFiber (EK1521)^Reused (EK1501)^Term 124 (EL1809) A4^Channel 12^Input} *)
	STP.P402A_JockeyPumpA_OnOffStat AT %IX137.1 : BOOL;	(*  ~ {LinkedWith:TIID^C6920 (EtherCAT)^ScadaRoom_KouplerUTP (EK1100)^ScadaRoom_KouplerFiber (EK1521)^Reused (EK1501)^Term 124 (EL1809) A4^Channel 13^Input} *)
	STP.P402B_JockeyPumpB_OnOffStat AT %IX137.2 : BOOL;	(*  ~ {LinkedWith:TIID^C6920 (EtherCAT)^ScadaRoom_KouplerUTP (EK1100)^ScadaRoom_KouplerFiber (EK1521)^Reused (EK1501)^Term 124 (EL1809) A4^Channel 14^Input} *)
	STP.P403A_VacuumPumpA_OnOffStat AT %IX137.3 : BOOL;	(*  ~ {LinkedWith:TIID^C6920 (EtherCAT)^ScadaRoom_KouplerUTP (EK1100)^ScadaRoom_KouplerFiber (EK1521)^Reused (EK1501)^Term 124 (EL1809) A4^Channel 15^Input} *)
	STP.P403B_VacuumPumpB_OnOffStat AT %IX137.4 : BOOL;	(*  ~ {LinkedWith:TIID^C6920 (EtherCAT)^ScadaRoom_KouplerUTP (EK1100)^ScadaRoom_KouplerFiber (EK1521)^Reused (EK1501)^Term 124 (EL1809) A4^Channel 16^Input} *)
	STP.P401A_LeadPumpA_EStopStat AT %IX137.5 : BOOL;	(*  ~ {LinkedWith:TIID^C6920 (EtherCAT)^ScadaRoom_KouplerUTP (EK1100)^ScadaRoom_KouplerFiber (EK1521)^Reused (EK1501)^Term 125 (EL1809) A5^Channel 1^Input} *)
	STP.P401B_LeadPumpB_EStopStat AT %IX137.6 : BOOL;	(*  ~ {LinkedWith:TIID^C6920 (EtherCAT)^ScadaRoom_KouplerUTP (EK1100)^ScadaRoom_KouplerFiber (EK1521)^Reused (EK1501)^Term 125 (EL1809) A5^Channel 2^Input} *)
	STP.P401C_LeadPumpC_EStopStat AT %IX137.7 : BOOL;	(*  ~ {LinkedWith:TIID^C6920 (EtherCAT)^ScadaRoom_KouplerUTP (EK1100)^ScadaRoom_KouplerFiber (EK1521)^Reused (EK1501)^Term 125 (EL1809) A5^Channel 3^Input} *)
	STP.P401D_LeadPumpD_EStopStat AT %IX138.0 : BOOL;	(*  ~ {LinkedWith:TIID^C6920 (EtherCAT)^ScadaRoom_KouplerUTP (EK1100)^ScadaRoom_KouplerFiber (EK1521)^Reused (EK1501)^Term 125 (EL1809) A5^Channel 4^Input} *)
	STP.P402A_JockeyPumpA_EStopStat AT %IX138.1 : BOOL;	(*  ~ {LinkedWith:TIID^C6920 (EtherCAT)^ScadaRoom_KouplerUTP (EK1100)^ScadaRoom_KouplerFiber (EK1521)^Reused (EK1501)^Term 125 (EL1809) A5^Channel 5^Input} *)
	STP.P402B_JockeyPumpB_EStopStat AT %IX138.2 : BOOL;	(*  ~ {LinkedWith:TIID^C6920 (EtherCAT)^ScadaRoom_KouplerUTP (EK1100)^ScadaRoom_KouplerFiber (EK1521)^Reused (EK1501)^Term 125 (EL1809) A5^Channel 6^Input} *)
	STP.P403A_VacuumPumpA_EStopStat AT %IX138.3 : BOOL;	(*  ~ {LinkedWith:TIID^C6920 (EtherCAT)^ScadaRoom_KouplerUTP (EK1100)^ScadaRoom_KouplerFiber (EK1521)^Reused (EK1501)^Term 125 (EL1809) A5^Channel 7^Input} *)
	STP.P403B_VacuumPumpB_EStopStat AT %IX138.4 : BOOL;	(*  ~ {LinkedWith:TIID^C6920 (EtherCAT)^ScadaRoom_KouplerUTP (EK1100)^ScadaRoom_KouplerFiber (EK1521)^Reused (EK1501)^Term 125 (EL1809) A5^Channel 8^Input} *)
	STP.XV401_SolenoidValve_OpenCmd AT %QX65.5 : BOOL;	(*  ~ {LinkedWith:TIID^C6920 (EtherCAT)^ScadaRoom_KouplerUTP (EK1100)^ScadaRoom_KouplerFiber (EK1521)^Reused (EK1501)^Term 126 (EL2809) A6^Channel 1^Output} *)
	STP.P401A_LeadPumpA_RunCmd AT %QX74.1 : BOOL;	(*  ~ {LinkedWith:TIID^C6920 (EtherCAT)^ScadaRoom_KouplerUTP (EK1100)^ScadaRoom_KouplerFiber (EK1521)^Reused (EK1501)^Term 126 (EL2809) A6^Channel 2^Output} *)
	STP.P401B_LeadPumpB_RunCmd AT %QX65.6 : BOOL;	(*  ~ {LinkedWith:TIID^C6920 (EtherCAT)^ScadaRoom_KouplerUTP (EK1100)^ScadaRoom_KouplerFiber (EK1521)^Reused (EK1501)^Term 126 (EL2809) A6^Channel 3^Output} *)
	STP.P401C_LeadPumpC_RunCmd AT %QX65.7 : BOOL;	(*  ~ {LinkedWith:TIID^C6920 (EtherCAT)^ScadaRoom_KouplerUTP (EK1100)^ScadaRoom_KouplerFiber (EK1521)^Reused (EK1501)^Term 126 (EL2809) A6^Channel 4^Output} *)
	STP.P401D_LeadPumpD_RunCmd AT %QX66.0 : BOOL;	(*  ~ {LinkedWith:TIID^C6920 (EtherCAT)^ScadaRoom_KouplerUTP (EK1100)^ScadaRoom_KouplerFiber (EK1521)^Reused (EK1501)^Term 126 (EL2809) A6^Channel 5^Output} *)
	STP.P402A_JockeyPumpA_RunCmd AT %QX66.1 : BOOL;	(*  ~ {LinkedWith:TIID^C6920 (EtherCAT)^ScadaRoom_KouplerUTP (EK1100)^ScadaRoom_KouplerFiber (EK1521)^Reused (EK1501)^Term 126 (EL2809) A6^Channel 6^Output} *)
	STP.P402B_JockeyPumpB_RunCmd AT %QX66.2 : BOOL;	(*  ~ {LinkedWith:TIID^C6920 (EtherCAT)^ScadaRoom_KouplerUTP (EK1100)^ScadaRoom_KouplerFiber (EK1521)^Reused (EK1501)^Term 126 (EL2809) A6^Channel 7^Output} *)
	STP.P403A_VacuumPumpA_RunCmd AT %QX66.3 : BOOL;	(*  ~ {LinkedWith:TIID^C6920 (EtherCAT)^ScadaRoom_KouplerUTP (EK1100)^ScadaRoom_KouplerFiber (EK1521)^Reused (EK1501)^Term 126 (EL2809) A6^Channel 8^Output} *)
	STP.P403B_VacuumPumpB_RunCmd AT %QX66.4 : BOOL;	(*  ~ {LinkedWith:TIID^C6920 (EtherCAT)^ScadaRoom_KouplerUTP (EK1100)^ScadaRoom_KouplerFiber (EK1521)^Reused (EK1501)^Term 126 (EL2809) A6^Channel 9^Output} *)
	STP.AUX415_AuxLamp_LowPressure AT %QX66.5 : BOOL;	(*  ~ {LinkedWith:TIID^C6920 (EtherCAT)^ScadaRoom_KouplerUTP (EK1100)^ScadaRoom_KouplerFiber (EK1521)^Reused (EK1501)^Term 126 (EL2809) A6^Channel 10^Output} *)
	STP.AUX416_AuxLamp_TankHighLevel AT %QX66.6 : BOOL;	(*  ~ {LinkedWith:TIID^C6920 (EtherCAT)^ScadaRoom_KouplerUTP (EK1100)^ScadaRoom_KouplerFiber (EK1521)^Reused (EK1501)^Term 126 (EL2809) A6^Channel 11^Output} *)
	STP.AUX417_AuxLamp_SystemPrimed AT %QX66.7 : BOOL;	(*  ~ {LinkedWith:TIID^C6920 (EtherCAT)^ScadaRoom_KouplerUTP (EK1100)^ScadaRoom_KouplerFiber (EK1521)^Reused (EK1501)^Term 126 (EL2809) A6^Channel 12^Output} *)
	STP.AUX801_CommonAlarm AT %QX74.2 : BOOL;	(*  ~ {LinkedWith:TIID^C6920 (EtherCAT)^ScadaRoom_KouplerUTP (EK1100)^ScadaRoom_KouplerFiber (EK1521)^Reused (EK1501)^Term 126 (EL2809) A6^Channel 13^Output} *)
	STP.AUX802_PLCRunStat AT %QX92.0 : BOOL;	(*  ~ {LinkedWith:TIID^C6920 (EtherCAT)^ScadaRoom_KouplerUTP (EK1100)^ScadaRoom_KouplerFiber (EK1521)^Reused (EK1501)^Term 126 (EL2809) A6^Channel 14^Output} *)
	STP.PSL411_PressureTransmitter_ScaledValue AT %IB546 : INT;	(*  ~ {LinkedWith:TIID^C6920 (EtherCAT)^ScadaRoom_KouplerUTP (EK1100)^ScadaRoom_KouplerFiber (EK1521)^Reused (EK1501)^Term 127 (EL3154) A7^AI Standard Channel 1^Value} *)
	STP.F900_FanStatus AT %IX300.0 : BOOL;	(*  ~ {LinkedWith:TIID^C6920 (EtherCAT)^ScadaRoom_KouplerUTP (EK1100)^ScadaRoom_KouplerFiber (EK1521)^ScadaRoom_KouplerFiber_Return (EK1501)^Term 129 (EL1088) A2^Channel 3^Input} *)
	STP.D900_DoorPanelStatus AT %IX460.0 : BOOL;	(*  ~ {LinkedWith:TIID^C6920 (EtherCAT)^ScadaRoom_KouplerUTP (EK1100)^ScadaRoom_KouplerFiber (EK1521)^ScadaRoom_KouplerFiber_Return (EK1501)^Term 129 (EL1088) A2^Channel 1^Input} *)
	STP.GENRUN_Generator_RunStat AT %IX300.2 : BOOL;	(*  ~ {LinkedWith:TIID^C6920 (EtherCAT)^ScadaRoom_KouplerUTP (EK1100)^ScadaRoom_KouplerFiber (EK1521)^ScadaRoom_KouplerFiber_Return (EK1501)^Term 129 (EL1088) A2^Channel 5^Input} *)
	STP.GENOT_Generator_OverloadStat AT %IX300.3 : BOOL;	(*  ~ {LinkedWith:TIID^C6920 (EtherCAT)^ScadaRoom_KouplerUTP (EK1100)^ScadaRoom_KouplerFiber (EK1521)^ScadaRoom_KouplerFiber_Return (EK1501)^Term 129 (EL1088) A2^Channel 7^Input} *)
	STP.GENFAIL_Generator_FailStat AT %IX300.4 : BOOL;	(*  ~ {LinkedWith:TIID^C6920 (EtherCAT)^ScadaRoom_KouplerUTP (EK1100)^ScadaRoom_KouplerFiber (EK1521)^ScadaRoom_KouplerFiber_Return (EK1501)^Term 129 (EL1088) A2^Channel 2^Input} *)
	STP.GENESTOP_Generator_EStop_Stat AT %IX480.0 : BOOL;	(*  ~ {LinkedWith:TIID^C6920 (EtherCAT)^ScadaRoom_KouplerUTP (EK1100)^ScadaRoom_KouplerFiber (EK1521)^ScadaRoom_KouplerFiber_Return (EK1501)^Term 129 (EL1088) A2^Channel 4^Input} *)
	STP.AUX902_PLCRunStat AT %QX92.1 : BOOL;	(*  ~ {LinkedWith:TIID^C6920 (EtherCAT)^ScadaRoom_KouplerUTP (EK1100)^ScadaRoom_KouplerFiber (EK1521)^ScadaRoom_KouplerFiber_Return (EK1501)^Term 130 (EL2809) A3^Channel 1^Output} *)
	STP.AUX901_CommonAlarm AT %QX84.1 : BOOL;	(*  ~ {LinkedWith:TIID^C6920 (EtherCAT)^ScadaRoom_KouplerUTP (EK1100)^ScadaRoom_KouplerFiber (EK1521)^ScadaRoom_KouplerFiber_Return (EK1501)^Term 130 (EL2809) A3^Channel 2^Output} *)
	STP.AUX903_GeneratorSupplyStat AT %QX84.2 : BOOL;	(*  ~ {LinkedWith:TIID^C6920 (EtherCAT)^ScadaRoom_KouplerUTP (EK1100)^ScadaRoom_KouplerFiber (EK1521)^ScadaRoom_KouplerFiber_Return (EK1501)^Term 130 (EL2809) A3^Channel 3^Output} *)
	STP.AUX904_Stream1_RunStat AT %QX84.3 : BOOL;	(*  ~ {LinkedWith:TIID^C6920 (EtherCAT)^ScadaRoom_KouplerUTP (EK1100)^ScadaRoom_KouplerFiber (EK1521)^ScadaRoom_KouplerFiber_Return (EK1501)^Term 130 (EL2809) A3^Channel 4^Output} *)
	STP.AUX905_Stream2_RunStat AT %QX84.4 : BOOL;	(*  ~ {LinkedWith:TIID^C6920 (EtherCAT)^ScadaRoom_KouplerUTP (EK1100)^ScadaRoom_KouplerFiber (EK1521)^ScadaRoom_KouplerFiber_Return (EK1501)^Term 130 (EL2809) A3^Channel 5^Output} *)
	STP.AUX906_InletWork1_RunStat AT %QX84.5 : BOOL;	(*  ~ {LinkedWith:TIID^C6920 (EtherCAT)^ScadaRoom_KouplerUTP (EK1100)^ScadaRoom_KouplerFiber (EK1521)^ScadaRoom_KouplerFiber_Return (EK1501)^Term 130 (EL2809) A3^Channel 6^Output} *)
	STP.AUX907_BlowerHouse1_RunStat AT %QX84.6 : BOOL;	(*  ~ {LinkedWith:TIID^C6920 (EtherCAT)^ScadaRoom_KouplerUTP (EK1100)^ScadaRoom_KouplerFiber (EK1521)^ScadaRoom_KouplerFiber_Return (EK1501)^Term 130 (EL2809) A3^Channel 7^Output} *)
	STP.AUX908_SBR1_RunStat AT %QX84.7 : BOOL;	(*  ~ {LinkedWith:TIID^C6920 (EtherCAT)^ScadaRoom_KouplerUTP (EK1100)^ScadaRoom_KouplerFiber (EK1521)^ScadaRoom_KouplerFiber_Return (EK1501)^Term 130 (EL2809) A3^Channel 8^Output} *)
	STP.AUX909_InletWork2_RunStat AT %QX85.0 : BOOL;	(*  ~ {LinkedWith:TIID^C6920 (EtherCAT)^ScadaRoom_KouplerUTP (EK1100)^ScadaRoom_KouplerFiber (EK1521)^ScadaRoom_KouplerFiber_Return (EK1501)^Term 130 (EL2809) A3^Channel 9^Output} *)
	STP.AUX910_BlowerHouse2_RunStat AT %QX85.1 : BOOL;	(*  ~ {LinkedWith:TIID^C6920 (EtherCAT)^ScadaRoom_KouplerUTP (EK1100)^ScadaRoom_KouplerFiber (EK1521)^ScadaRoom_KouplerFiber_Return (EK1501)^Term 130 (EL2809) A3^Channel 10^Output} *)
	STP.AUX911_SBR2_RunStat AT %QX85.2 : BOOL;	(*  ~ {LinkedWith:TIID^C6920 (EtherCAT)^ScadaRoom_KouplerUTP (EK1100)^ScadaRoom_KouplerFiber (EK1521)^ScadaRoom_KouplerFiber_Return (EK1501)^Term 130 (EL2809) A3^Channel 11^Output} *)
	STP.AUX912_ChemicalTertiary_RunStat AT %QX85.3 : BOOL;	(*  ~ {LinkedWith:TIID^C6920 (EtherCAT)^ScadaRoom_KouplerUTP (EK1100)^ScadaRoom_KouplerFiber (EK1521)^ScadaRoom_KouplerFiber_Return (EK1501)^Term 130 (EL2809) A3^Channel 12^Output} *)
	STP.AUX913_SludgeThickening_RunStat AT %QX85.4 : BOOL;	(*  ~ {LinkedWith:TIID^C6920 (EtherCAT)^ScadaRoom_KouplerUTP (EK1100)^ScadaRoom_KouplerFiber (EK1521)^ScadaRoom_KouplerFiber_Return (EK1501)^Term 130 (EL2809) A3^Channel 13^Output} *)
	STP.AUX914_FilterPress_RunStat AT %QX85.5 : BOOL;	(*  ~ {LinkedWith:TIID^C6920 (EtherCAT)^ScadaRoom_KouplerUTP (EK1100)^ScadaRoom_KouplerFiber (EK1521)^ScadaRoom_KouplerFiber_Return (EK1501)^Term 130 (EL2809) A3^Channel 14^Output} *)
	STP.AUX915_Reuse_RunStat AT %QX85.6 : BOOL;	(*  ~ {LinkedWith:TIID^C6920 (EtherCAT)^ScadaRoom_KouplerUTP (EK1100)^ScadaRoom_KouplerFiber (EK1521)^ScadaRoom_KouplerFiber_Return (EK1501)^Term 130 (EL2809) A3^Channel 15^Output} *)
	STP.ScadaRoom_KouplerUTP_State AT %IB304 : UINT;	(*  ~ {LinkedWith:TIID^C6920 (EtherCAT)^ScadaRoom_KouplerUTP (EK1100)^InfoData^State} *)
	STP.ScadaRoom_KouplerFiber_State AT %IB306 : UINT;	(*  ~ {LinkedWith:TIID^C6920 (EtherCAT)^ScadaRoom_KouplerUTP (EK1100)^ScadaRoom_KouplerFiber (EK1521)^InfoData^State} *)
	STP.InletWork_1_KouplerFiber_State AT %IB308 : UINT;	(*  ~ {LinkedWith:TIID^C6920 (EtherCAT)^ScadaRoom_KouplerUTP (EK1100)^ScadaRoom_KouplerFiber (EK1521)^InletWork_1(EK1501)^InfoData^State} *)
	STP.InletWork_2_KouplerFiber_State AT %IB310 : UINT;	(*  ~ {LinkedWith:TIID^C6920 (EtherCAT)^ScadaRoom_KouplerUTP (EK1100)^ScadaRoom_KouplerFiber (EK1521)^InletWork_1(EK1501)^InletWork_2 (EK1122)^InfoData^State} *)
	STP.BlowerHouse_2_KouplerFiber_State AT %IB312 : UINT;	(*  ~ {LinkedWith:TIID^C6920 (EtherCAT)^ScadaRoom_KouplerUTP (EK1100)^ScadaRoom_KouplerFiber (EK1521)^BlowerHouse_2 (EK1501)^InfoData^State} *)
	STP.BlowerHouse_1_KouplerFiber_State AT %IB314 : UINT;	(*  ~ {LinkedWith:TIID^C6920 (EtherCAT)^ScadaRoom_KouplerUTP (EK1100)^ScadaRoom_KouplerFiber (EK1521)^BlowerHouse_2 (EK1501)^BlowerHouse_1 (EK1122)^InfoData^State} *)
	STP.SBR_1_KouplerFiber_State AT %IB316 : UINT;	(*  ~ {LinkedWith:TIID^C6920 (EtherCAT)^ScadaRoom_KouplerUTP (EK1100)^ScadaRoom_KouplerFiber (EK1521)^SBR_1 (EK1501)^InfoData^State} *)
	STP.SBR_2_KouplerFiber_State AT %IB318 : UINT;	(*  ~ {LinkedWith:TIID^C6920 (EtherCAT)^ScadaRoom_KouplerUTP (EK1100)^ScadaRoom_KouplerFiber (EK1521)^SBR_2 (EK1501)^InfoData^State} *)
	STP.ChemicalAndTertiary_KouplerFiber_State AT %IB320 : UINT;	(*  ~ {LinkedWith:TIID^C6920 (EtherCAT)^ScadaRoom_KouplerUTP (EK1100)^ScadaRoom_KouplerFiber (EK1521)^ChemicalAndTertiary (EK1501)^InfoData^State} *)
	STP.ChemicalAndTertiary_KouplerUTP_State AT %IB476 : UINT;	(*  ~ {LinkedWith:TIID^C6920 (EtherCAT)^ScadaRoom_KouplerUTP (EK1100)^ScadaRoom_KouplerFiber (EK1521)^ChemicalAndTertiary (EK1501)^Term 96 (EK1122)^InfoData^State} *)
	STP.SludgeThickening_KouplerFiber_State AT %IB322 : UINT;	(*  ~ {LinkedWith:TIID^C6920 (EtherCAT)^ScadaRoom_KouplerUTP (EK1100)^ScadaRoom_KouplerFiber (EK1521)^SludgeThickening (EK1501)^InfoData^State} *)
	STP.Reused_KouplerFiber_State AT %IB324 : UINT;	(*  ~ {LinkedWith:TIID^C6920 (EtherCAT)^ScadaRoom_KouplerUTP (EK1100)^ScadaRoom_KouplerFiber (EK1521)^Reused (EK1501)^InfoData^State} *)
	STP.ScadaRoom_KouplerFiber_Return_State AT %IB326 : UINT;	(*  ~ {LinkedWith:TIID^C6920 (EtherCAT)^ScadaRoom_KouplerUTP (EK1100)^ScadaRoom_KouplerFiber (EK1521)^ScadaRoom_KouplerFiber_Return (EK1501)^InfoData^State} *)
	STP.RST001A_ResetButtonInlet_1 AT %IX472.0 : BOOL;	(*  ~ {LinkedWith:TIID^C6920 (EtherCAT)^ScadaRoom_KouplerUTP (EK1100)^ScadaRoom_KouplerFiber (EK1521)^InletWork_1(EK1501)^Term 12 (EL1809) A9^Channel 12^Input} *)
	STP.RST001B_ResetButtonInlet_2 AT %IX472.1 : BOOL;	(*  ~ {LinkedWith:TIID^C6920 (EtherCAT)^ScadaRoom_KouplerUTP (EK1100)^ScadaRoom_KouplerFiber (EK1521)^InletWork_1(EK1501)^Term 12 (EL1809) A9^Channel 13^Input} *)
	STP.RST002A_ResetButtonBlowerHouse_1 AT %IX472.2 : BOOL;	(*  ~ {LinkedWith:TIID^C6920 (EtherCAT)^ScadaRoom_KouplerUTP (EK1100)^ScadaRoom_KouplerFiber (EK1521)^BlowerHouse_2 (EK1501)^BlowerHouse_1 (EK1122)^Term 42 (EK1100)^Term 51 (EL1809) A10^Channel 9^Input} *)
	STP.RST002B_ResetButtonBlowerHouse_2 AT %IX472.3 : BOOL;	(*  ~ {LinkedWith:TIID^C6920 (EtherCAT)^ScadaRoom_KouplerUTP (EK1100)^ScadaRoom_KouplerFiber (EK1521)^BlowerHouse_2 (EK1501)^Term 37 (EL1809) A25^Channel 9^Input} *)
	STP.RST003A_ResetButtonSBR_1 AT %IX472.4 : BOOL;	(*  ~ {LinkedWith:TIID^C6920 (EtherCAT)^ScadaRoom_KouplerUTP (EK1100)^ScadaRoom_KouplerFiber (EK1521)^SBR_1 (EK1501)^Term 61 (EL1809) A6^Channel 9^Input} *)
	STP.RST003B_ResetButtonSBR_2 AT %IX478.0 : BOOL;	(*  ~ {LinkedWith:TIID^C6920 (EtherCAT)^ScadaRoom_KouplerUTP (EK1100)^ScadaRoom_KouplerFiber (EK1521)^SBR_2 (EK1501)^Term 74 (EL1809) A6^Channel 9^Input} *)
	STP.RST004_ResetButtonChemicalTertiary AT %IX472.6 : BOOL;	(*  ~ {LinkedWith:TIID^C6920 (EtherCAT)^ScadaRoom_KouplerUTP (EK1100)^ScadaRoom_KouplerFiber (EK1521)^ChemicalAndTertiary (EK1501)^Term 95 (EL1809) A14^Channel 14^Input} *)
	STP.RST005_ResetButtonSludgeThickening AT %IX478.1 : BOOL;	(*  ~ {LinkedWith:TIID^C6920 (EtherCAT)^ScadaRoom_KouplerUTP (EK1100)^ScadaRoom_KouplerFiber (EK1521)^SludgeThickening (EK1501)^Term 116 (EL1809) A10^Channel 15^Input} *)
	STP.RST008_ResetButtonReused AT %IX473.2 : BOOL;	(*  ~ {LinkedWith:TIID^C6920 (EtherCAT)^ScadaRoom_KouplerUTP (EK1100)^ScadaRoom_KouplerFiber (EK1521)^Reused (EK1501)^Term 125 (EL1809) A5^Channel 15^Input} *)
	STP.sbr_reset_A1 AT %IX548.0 : BOOL;
	STP.sbr_reset_A2 AT %IX548.1 : BOOL;
	STP.sbr_reset_A3 AT %IX548.2 : BOOL;
	STP.sbr_reset_A4 AT %IX548.3 : BOOL;
	STP.sbr_reset_B1 AT %IX548.4 : BOOL;
	STP.sbr_reset_B2 AT %IX548.5 : BOOL;
	STP.sbr_reset_B3 AT %IX548.6 : BOOL;
	STP.sbr_reset_B4 AT %IX548.7 : BOOL;
END_VAR

